// ---- VISUs/GlobalTextList_1.TcGTLO
TEXTLIST GlobalTextList_1
  2681 = '     '
  119 = '%' | German: '%' | France: '%' | English: '%'
  1446 = '%0.01f' | German: '%0.01f' | France: '%0.01f' | English: '%0.01f'
  4503 = '%0.02f' | German: '%0.02f' | France: '%0.02f' | English: '%0.02f'
  2738 = '%0.1f' | German: '%0.1f' | France: '%0.1f' | English: '%0.1f'
  537 = '%d' | German: '%d' | France: '%d' | English: '%d'
  890 = '%i' | German: '%i' | France: '%i' | English: '%i'
  1226 = '%i0.01f' | German: '%i0.01f' | France: '%i0.01f' | English: '%i0.01f'
  889 = '%s' | German: '%s' | France: '%s' | English: '%s'
  2909 = '(X100.00) STN 01 - 03 ULTRASONIC GENERATOR MCB - TRIP (-10F1)\n' | German: '(X100.00) WANNE 01 - WANNE 03 ULTRASCHALL GENERATOR SICHERUNG A AUSGELÖST (-10F1)' | France: '(X100.00) DEFAUT DISJONCTEUR GENE US POS 1 - POS 3 (-10F1)' | English: '(X100.00) STN 01 - 03 ULTRASONIC GENERATOR MCB - TRIP (-10F1)\n'
  3104 = '(X100.01) STN 01 ULTRASONIC GENERATOR (LEFT & RIGHT) - ALARM (-10U1)' | German: '(X100.01) WANNE 01 ULTRASCHALL GENERATOR (SEITE) SICHERUNG AUSGELÖST (-10U1)' | France: '(X100.01) CUVE 1 ALARME DU GENERATEUR ULTRASONS (COTE) (-10U1)' | English: '(X100.01) STN 01 ULTRASONIC GENERATOR (LEFT & RIGHT) - ALARM (-10U1)'
  9404 = '(X100.02) STN 01 ULTRASONIC GENERATOR (BOTTOM) - ALARM (-10U1)\n' | German: '(X100.02) WANNE 01 ULTRASCHALL GENERATOR (UNTEN) SICHERUNG AUSGELÖST (-10U1)' | France: '(X100.02) CUVE 2 ALARME DU GENERATEUR ULTRASONS (FOND) (-10U1)' | English: '(X100.02) STN 01 ULTRASONIC GENERATOR (BOTTOM) - ALARM (-10U1)\n'
  10481 = '(X100.03) STN 02 ULTRASONIC GENERATOR (LEFT & RIGHT) - ALARM (-10U1)\n' | German: '(X100.03) WANNE 02 ULTRASCHALL GENERATOR (SEITE) SICHERUNG AUSGELÖST (-10U1)' | France: '(X100.03) CUVE 2 ALARME DU GENERATEUR ULTRASONS (COTE) (-10U1)' | English: '(X100.03) STN 02 ULTRASONIC GENERATOR (LEFT & RIGHT) - ALARM (-10U1)\n'
  10488 = '(X100.04) STN 02 ULTRASONIC GENERATOR (BOTTOM) - ALARM (-10U1)\n' | German: '(X100.04) WANNE 02 ULTRASCHALL GENERATOR (UNTEN) SICHERUNG AUSGELÖST (-10U1)' | France: '(X100.04) CUVE 2 ALARME DU GENERATEUR ULTRASONS (FOND) (-10U1)' | English: '(X100.04) STN 02 ULTRASONIC GENERATOR (BOTTOM) - ALARM (-10U1)\n'
  5247 = '(X100.05) STN 03 ULTRASONIC GENERATOR (LEFT & RIGHT) - ALARM (-10U1)' | German: '(X100.05) WANNE 03 ULTRASCHALL GENERATOR (SEITE) SICHERUNG AUSGELÖST (-10U1)' | France: '(X100.05) CUVE 3 ALARME DU GENERATEUR ULTRASONS (COTE) (-10U1)' | English: '(X100.05) STN 03 ULTRASONIC GENERATOR (LEFT & RIGHT) - ALARM (-10U1)'
  11591 = '(X100.06) STN 03 ULTRASONIC GENERATOR (BOTTOM) - ALARM (-10U1)' | German: '(X100.06) WANNE 03 ULTRASCHALL GENERATOR (UNTEN) SICHERUNG AUSGELÖST (-10U1)' | France: '(X100.06) CUVE 3 ALARME DU GENERATEUR ULTRASONS (FOND) (-10U1)' | English: '(X100.06) STN 03 ULTRASONIC GENERATOR (BOTTOM) - ALARM (-10U1)'
  12139 = '(X100.07) STN 04 - 05 ULTRASONIC GENERATOR MCB - TRIP (-11F1)' | German: '(X100.07) WANNE 04 - WANNE 05 ULTRASCHALL GENERATOR SICHERUNG AUSGELÖST (-11F1)' | France: '(X100.07) DEFAUT DISJONCTEUR GENE US CUVE 4 - CUVE 5 (-11F1)' | English: '(X100.07) STN 04 - 05 ULTRASONIC GENERATOR MCB - TRIP (-11F1)'
  6933 = '(X100.08) STN 04 ULTRASONIC GENERATOR (LEFT & RIGHT) - ALARM (-11U1)' | German: '(X100.08) WANNE 04 ULTRASCHALL GENERATOR (SEITE) SICHERUNG AUSGELÖST (-11U1)' | France: '(X100.08) CUVE 4 ALARME DU GENERATEUR ULTRASONS (COTE) (-11U1)' | English: '(X100.08) STN 04 ULTRASONIC GENERATOR (LEFT & RIGHT) - ALARM (-11U1)'
  6619 = '(X100.09) STN 04 ULTRASONIC GENERATOR (BOTTOM) - ALARM (-11U1)' | German: '(X100.09) WANNE 04 ULTRASCHALL GENERATOR (UNTEN) SICHERUNG AUSGELÖST (-11U1)' | France: '(X100.09) CUVE 4 ALARME DU GENERATEUR ULTRASONS (FOND) (-11U1)' | English: '(X100.09) STN 04 ULTRASONIC GENERATOR (BOTTOM) - ALARM (-11U1)'
  4361 = '(X100.10) STN 05 ULTRASONIC GENERATOR (BOTTOM) - ALARM (-11U1)' | German: '(X100.10) WANNE 05 ULTRASCHALL GENERATOR (UNTEN) SICHERUNG AUSGELÖST (-11U1)' | France: '(X100.10) CUVE 5 ALARME DU GENERATEUR ULTRASONS (FOND) (-11U1)' | English: '(X100.10) STN 05 ULTRASONIC GENERATOR (BOTTOM) - ALARM (-11U1)'
  1199 = '(X100.11) GENERAL MAIN PANEL PB - E-STOP (-251S1)' | German: '(X100.11) HAUPTPANEL - NOT-AUS (-251S1)' | France: "(X100.11) ALARME ARRET D'URGENCE - BP PANEL (-251S1)" | English: '(X100.11) GENERAL MAIN PANEL PB - E-STOP (-251S1)'
  10185 = '(X100.12) OPERATOR PULL STRING - E-STOP (-251S2)' | German: '(X100.12) SICHERHEITSSEILZUG - NOT-AUS (-251S2)' | France: '(X100.12) DEFAUT BOUCLE ARRET URGENCE (-251S2)' | English: '(X100.12) OPERATOR PULL STRING - E-STOP (-251S2)'
  10087 = '(X100.13) MAINTENANCE PULL STRING - E-STOP  (-251S3)' | German: '(X100.13)WARTUNGSEILZUG NOT-AUS(-251S3)' | France: "(X100.13) CORDE D'ENTRETIEN - ARRÊT D'URGENCE (-251S3)" | English: '(X100.13) MAINTENANCE PULL STRING - E-STOP  (-251S3)'
  6489 = '(X100.14) GENERAL TOUCH MONITOR SOCKET ELCB - TRIP (-8Q1)' | German: '(X100.14) TOUCH SCREEN STECKDOSE SICHERUNG AUSGELÖST (-8Q1)' | France: '(X100.14) DEFAUT DISJONCTEUR PANEL OPERATEUR (-8Q1)' | English: '(X100.14) GENERAL TOUCH MONITOR SOCKET ELCB - TRIP (-8Q1)'
  7510 = '(X100.15) ARM 01 SERVO DRIVE MCB - TRIP (-40F1)' | German: '(X100.15) ARM 01 SERVO ANTRIEB MCB - AUSLÖSUNG (-40F1)' | France: '(X100.15) DEFAUT DISJONCTEUR SERVOMOTEUR ROBOT (-40F1)' | English: '(X100.15) ARM 01 SERVO DRIVE MCB - TRIP (-40F1)'
  11212 = '(X101.00) IPC DC ON SIGNAL (-410K1)' | German: '(X101.00) INDUSTRIE-PC GLEICHSTROM AUF SIGNAL (-410K1)' | France: '(X101.00)PC INDUSTRIEL COURANT CONTINU SUR SIGNAL(-410K1)' | English: '(X101.00) IPC DC ON SIGNAL (-410K1)'
  2968 = '(X101.01) PANEL VENTILATION FAN MCB - TRIP  (-6F1)\n' | German: '(X101.01) SCHALTSCHRANK VENTILATOR SICHERUNG AUSGELÖST  (-6F1)' | France: '(X101.01) DEFAUT DISJONCTEUR VENTILATEUR ARMOIRE ELECTRIQUE  (-6F1)' | English: '(X101.01) PANEL VENTILATION FAN MCB - TRIP  (-6F1)\n'
  9585 = '(X101.02) PANEL LIGHTING MCB - TRIP  (-5F1)' | German: '(X101.02) SCHALTSCHRANK BELEUCHTUNG SICHERUNG AUSGELÖST  (-5F1)' | France: '(X101.02) DEFAUT DISJONCTEUR ECLAIRAGE 1  (-5F1)' | English: '(X101.02) PANEL LIGHTING MCB - TRIP  (-5F1)'
  4159 = '(X101.03) MACHINE LIGHTING 01 MCB - TRIP (-5F2)' | German: '(X101.03) MASCHINENBELEUCHTUNG 01(-5F2)' | France: '(X101.03)ÉCLAIRAGE DE MACHINE 01(-5F2)' | English: '(X101.03) MACHINE LIGHTING 01 MCB - TRIP (-5F2)'
  7312 = '(X101.04) MACHINE LIGHTING 02 MCB - TRIP (-5F3)' | German: '(X101.04) MASCHINENBELEUCHTUNG 02(-5F3)' | France: '(X101.04)ÉCLAIRAGE DE MACHINE 02(-5F3)' | English: '(X101.04) MACHINE LIGHTING 02 MCB - TRIP (-5F3)'
  4346 = '(X101.05) GENERAL TOUCH MONITOR SOCKET MCB - TRIP (-8F1)' | German: '(X101.05) TOUCH SCREEN STECKDOSE SICHERUNG AUSGELÖST (-8F1)' | France: '(X101.05) DEFAUT DISJONCTEUR PANEL OPERATEUR (-8F1)' | English: '(X101.05) GENERAL TOUCH MONITOR SOCKET MCB - TRIP (-8F1)'
  8277 = '(X101.06) GENERAL PHASE SEQUENCE RELAY MCB - TRIP (-3F2)' | German: '(X101.06) DREHRICHTUNGSRELAIS SICHERUNG AUSGELÖST (-3F2)' | France: '(X101.06) DEFAUT DISJONCTEUR GENERAL (-3F2)' | English: '(X101.06) GENERAL PHASE SEQUENCE RELAY MCB - TRIP (-3F2)'
  9048 = '(X101.07) GENERAL PHASE SEQUENCE RELAY - TRIP (-3K1)' | German: '(X101.07) DREHRICHTUNGSRELAIS AUSGELÖST - ALARM (-3K1)' | France: '(X101.07) RELAIS ALARME  PHASE SEQUENCE (-3K1)' | English: '(X101.07) GENERAL PHASE SEQUENCE RELAY - TRIP (-3K1)'
  10253 = '(X101.08) STN 06 PROCESS TANK BLOWER MMS&TOR - TRIP (-100Q1)' | German: 'WANNE 06 PROZESS TANK GEBLÄSE MANUELLER MOTORSTARTER & THERMISCHE ÜBERLASTUNG AUSGELÖST' | France: 'CUVE 06 PROCESSUS RÉSERVOIR VENTILATEUR DÉMARRAGE MANUEL DU MOTEUR & SURCHARGE THERMIQUE DÉCLENCHÉE' | English: '(X101.08) STN 06 PROCESS TANK BLOWER MMS&TOR - TRIP (-100Q1)'
  5932 = '(X101.09) STN 01 - 06 EXHAUST BLOWER MMS&TOR - TRIP (-101Q1)' | German: 'WANNE 01 - 06 ABGASGEBLÄSE MANUELLER MOTORSTARTER & THERMISCHE ÜBERLASTUNG AUSGELÖST' | France: "CUVE 01 - 06 VENTILATEUR DE GAZ D'ÉCHAPPEMENT DÉMARRAGE MANUEL DU MOTEUR & SURCHARGE THERMIQUE DÉCLENCHÉE" | English: '(X101.09) STN 01 - 06 EXHAUST BLOWER MMS&TOR - TRIP (-101Q1)'
  6620 = '(X101.10) STN 01 - 05 AGITATION MOTOR MMS&TOR - TRIP (-160Q1)' | German: 'WANNE 01 - 05 MOTOR WARENBEWEGUNG MANUELLER MOTORSTARTER & THERMISCHE ÜBERLASTUNG AUSGELÖST' | France: 'CUVE 01 - 05 MOTEUR MOUVEMENT DU PRODUIT DÉMARREUR MANUEL DU MOTEUR & SURCHARGE THERMIQUE DÉCLENCHÉE' | English: '(X101.10) STN 01 - 05 AGITATION MOTOR MMS&TOR - TRIP (-160Q1)'
  5425 = '(X101.11) STN 01 DOSING PUMP MCB - TRIP (-70F1)' | German: '(X101.11) WANNE 01 DOSIERPUMPE SICHERUNG AUSGELÖST (-70F1)' | France: '(X101.11) CUVE 1 DEFAUT DISJONCTEUR POMPE DOSAGE (-70F1)' | English: '(X101.11) STN 01 DOSING PUMP MCB - TRIP (-70F1)'
  3137 = '(X101.12) STN 02 DOSING PUMP MCB - TRIP (-71F1)' | German: '(X101.12) WANNE 02 DOSIERPUMPE SICHERUNG AUSGELÖST (-71F1)' | France: '(X101.12) CUVE 2 DEFAUT DISJONCTEUR POMPE DOSAGE (-71F1)' | English: '(X101.12) STN 02 DOSING PUMP MCB - TRIP (-71F1)'
  3866 = '(X101.13) STN 03 DOSING PUMP MCB - TRIP (-72F1)' | German: '(X101.13) WANNE 03 DOSIERPUMPE SICHERUNG AUSGELÖST (-72F1)' | France: '(X101.13) CUVE 3 DEFAUT DISJONCTEUR POMPE DOSAGE (-72F1)' | English: '(X101.13) STN 03 DOSING PUMP MCB - TRIP (-72F1)'
  11364 = '(X101.14) STN 04 DOSING PUMP MCB - TRIP (-73F1)' | German: '(X101.14) WANNE 04 DOSIERPUMPE SICHERUNG AUSGELÖST (-73F1)' | France: '(X101.14) CUVE 4 DEFAUT DISJONCTEUR POMPE DOSAGE (-73F1)' | English: '(X101.14) STN 04 DOSING PUMP MCB - TRIP (-73F1)'
  8857 = '(X101.15) STN 01 DOSING CHEMICAL CONTAINER RELAY SIGNAL - FEEDBACK (-70K1)' | German: '(X101.15) WANNE 01 REINIGUNGSMITTELBEHÄLTER SENSOR 1 KONTAKTBLOCK - RÜCKMELDUNG (-70K1)' | France: '(X101.15) CUVE 1 DOSAGE RETOUR DU SIGNAL DU RELAIS DU CONTENEUR (-70K1)' | English: '(X101.15) STN 01 DOSING CHEMICAL CONTAINER RELAY SIGNAL - FEEDBACK (-70K1)'
  620 = '(X102.00) STN 01 PROCESS TANK PUMP MMS&TOR - TRIP (-74Q1)' | German: 'Wanne 01 Prozess Pumpe Tank Manueller Motorstarter & Thermische Überlastung Ausgelöst' | France: 'Cuve 01 Processus Pompe Réservoir Démarreur Manuel Du Moteur & Surcharge Thermique Déclenchée' | English: '(X102.00) STN 01 PROCESS TANK PUMP MMS&TOR - TRIP (-74Q1)'
  9751 = '(X102.01) STN 02 PROCESS TANK PUMP MMS&TOR - TRIP (-75Q1)' | German: 'Wanne 02 Prozess Pumpe Tank Manueller Motorstarter & Thermische Überlastung Ausgelöst' | France: 'Cuve 02 Processus Pompe Réservoir Démarreur Manuel Du Moteur & Surcharge Thermique Déclenchée' | English: '(X102.01) STN 02 PROCESS TANK PUMP MMS&TOR - TRIP (-75Q1)'
  11969 = '(X102.02) STN 03 PROCESS TANK PUMP MMS&TOR - TRIP (-76Q1)' | German: 'Wanne 03 Prozess Pumpe Tank Manueller Motorstarter & Thermische Überlastung Ausgelöst' | France: 'Cuve 03 Processus Pompe Réservoir Démarreur Manuel Du Moteur & Surcharge Thermique Déclenchée' | English: '(X102.02) STN 03 PROCESS TANK PUMP MMS&TOR - TRIP (-76Q1)'
  9673 = '(X102.03) STN 04 PROCESS TANK PUMP MMS&TOR - TRIP (-77Q1)' | German: 'Wanne 04 Prozess Pumpe Tank Manueller Motorstarter & Thermische Überlastung Ausgelöst' | France: 'Cuve 04 Processus Pompe Réservoir Démarreur Manuel Du Moteur & Surcharge Thermique Déclenchée' | English: '(X102.03) STN 04 PROCESS TANK PUMP MMS&TOR - TRIP (-77Q1)'
  4653 = '(X102.04) STN 05 PROCESS TANK PUMP MMS&TOR - TRIP (-78Q1)' | German: 'Wanne 05 Prozess Pumpe Tank Manueller Motorstarter & Thermische Überlastung Ausgelöst' | France: 'Cuve 05 Processus Pompe Réservoir Démarreur Manuel Du Moteur & Surcharge Thermique Déclenchée' | English: '(X102.04) STN 05 PROCESS TANK PUMP MMS&TOR - TRIP (-78Q1)'
  1689 = '(X102.05) STN 01 - 04 CHEMICAL RETURN TANK PUMP MMS&TOR - TRIP (-80Q1)' | German: 'Wanne 01 - 04 Pumpe Für Chemikalienrücklauftank Manueller Motoranlasser & Thermisches Überlastung Ausgelöst' | France: 'Cuve 01 - 04 Pompe Pour Réservoir De Retour De Produits Chimiques Démarreur Manuel Du Moteur & Relais Thermique De Surcharge Déclenché' | English: '(X102.05) STN 01 - 04 CHEMICAL RETURN TANK PUMP MMS&TOR - TRIP (-80Q1)'
  5529 = '(X102.06) STN 06 PROCESS TANK VACUUM PUMP MMS&TOR -TRIP (-79Q1)' | German: 'Wanne 06 Prozess Tank Vakuumpumpe Manueller Motorstarter & Thermische Überlastung Ausgelöst' | France: 'Cuve 06 Processus Réservoir Pompe À Vide Démarreur Manuel Du Moteur & Surcharge Thermique Déclenchée' | English: '(X102.06) STN 06 PROCESS TANK VACUUM PUMP MMS&TOR -TRIP (-79Q1)'
  315 = '(X102.07) STN 01 PROCESS TANK HEATER MCB - TRIP (-130F1)' | German: '(X102.07) WANNE 01 HEIZUNG SICHERUNG AUSGELÖST (-130F1)' | France: '(X102.07) CUVE 1 DEFAUT DISJONCTEUR CHAUFFAGE (-130F1)' | English: '(X102.07) STN 01 PROCESS TANK HEATER MCB - TRIP (-130F1)'
  910 = '(X102.08) STN 02 PROCESS TANK HEATER MCB - TRIP (-131F1)' | German: '(X102.08) WANNE 02 HEIZUNG SICHERUNG AUSGELÖST (-131F1)' | France: '(X102.08) CUVE 2 DEFAUT DISJONCTEUR CHAUFFAGE (-131F1)' | English: '(X102.08) STN 02 PROCESS TANK HEATER MCB - TRIP (-131F1)'
  6525 = '(X102.09) STN 03 PROCESS TANK HEATER MCB - TRIP (-132F1)' | German: '(X102.09) WANNE 03 HEIZUNG SICHERUNG AUSGELÖST (-132F1)' | France: '(X102.09) CUVE 3 DEFAUT DISJONCTEUR CHAUFFAGE (-132F1)' | English: '(X102.09) STN 03 PROCESS TANK HEATER MCB - TRIP (-132F1)'
  11585 = '(X102.10) STN 04 PROCESS TANK HEATER MCB - TRIP (-133F1)' | German: '(X102.10) WANNE 04 HEIZUNG SICHERUNG AUSGELÖST (-133F1)' | France: '(X102.10) CUVE 4 DEFAUT DISJONCTEUR CHAUFFAGE (-133F1)' | English: '(X102.10) STN 04 PROCESS TANK HEATER MCB - TRIP (-133F1)'
  3596 = '(X102.11) STN 06 PROCESS TANK HEATER MCB - TRIP (-134F1)' | German: '(X102.11) WANNE 06 HEIZUNG SICHERUNG AUSGELÖST (-134F1)' | France: '(X102.11) CUVE 6 DEFAUT DISJONCTEUR CHAUFFAGE (-134F1)' | English: '(X102.11) STN 06 PROCESS TANK HEATER MCB - TRIP (-134F1)'
  1057 = '(X102.12) LOADING CONVEYOR 1 MCB - TRIP (-170F1)' | German: '(X102.12) BELADEN FÖRDERBAND MOTOR 1 SICHERUNG AUSGELÖST (-170F1)' | France: '(X102.12) DISJONCTEUR CHARGEMENT MOTEUR CONV CHARG 1 (-170F1)' | English: '(X102.12) LOADING CONVEYOR 1 MCB - TRIP (-170F1)'
  11382 = '(X102.13) LOADING CONVEYOR 2 MCB - TRIP (-171F1)' | German: '(X102.13) BELADEN FÖRDERBAND MOTOR 2 SICHERUNG AUSGELÖST (-171F1)' | France: '(X102.13) DISJONCTEUR CHARGEMENT MOTEUR CONV CHARG 2 (-171F1)' | English: '(X102.13) LOADING CONVEYOR 2 MCB - TRIP (-171F1)'
  1453 = '(X102.14) LOADING CONVEYOR 3 MCB - TRIP (-172F1)' | German: '(X102.14) BELADEN FÖRDERBAND MOTOR 3 SICHERUNG AUSGELÖST (-172F1)' | France: '(X102.14) DISJONCTEUR CHARGEMENT MOTEUR CONV CHARG 3 (-172F1)' | English: '(X102.14) LOADING CONVEYOR 3 MCB - TRIP (-172F1)'
  1076 = '(X102.15) STN 02 DOSING CHEMICAL CONTAINER RELAY SIGNAL - FEEDBACK (-71K1)\n' | German: '(X102.15) WANNE 02 REINIGUNGSMITTELBEHÄLTER SENSOR 1 KONTAKTBLOCK - RÜCKMELDUNG (-71K1)' | France: '(X102.15) CUVE 2 DOSAGE RETOUR DU SIGNAL DU RELAIS DU CONTENEUR (-71K1)' | English: '(X102.15) STN 02 DOSING CHEMICAL CONTAINER RELAY SIGNAL - FEEDBACK (-71K1)\n'
  2864 = '(X103.00) MAIN SAFETY CONTACTOR 1 - FEEDBACK  (-250K1)' | German: '(X103.00) HAUPTSICHERHEITSSCHÜTZ 1 - RÜCKMELDUNG  (-250K1)' | France: '(X103.00) DEFAUT RETOUR CONTACTEUR GENERAL 1  (-250K1)' | English: '(X103.00) MAIN SAFETY CONTACTOR 1 - FEEDBACK  (-250K1)'
  3842 = '(X103.01) MAIN SAFETY CONTACTOR 2 - FEEDBACK  (-250K2)' | German: '(X103.01) HAUPTSICHERHEITSSCHÜTZ 2 - RÜCKMELDUNG  (-250K2)' | France: '(X103.01) DEFAUT RETOUR CONTACTEUR GENERAL 2  (-250K2)' | English: '(X103.01) MAIN SAFETY CONTACTOR 2 - FEEDBACK  (-250K2)'
  9985 = '(X103.02) DOOR SAFETY  CONTACTOR 1 - FEEDBACK  (-255K1)' | German: '(X103.02) TÜRSICHERHEITSSCHÜTZ 1 - RÜCKMELDUNG  (-255K1)' | France: '(X103.02) DEFAUT RETOUR CONTACTEUR SECURITE PORTE 1  (-255K1)' | English: '(X103.02) DOOR SAFETY  CONTACTOR 1 - FEEDBACK  (-255K1)'
  4912 = '(X103.03) DOOR SAFETY  CONTACTOR 2 - FEEDBACK  (-255K2)' | German: '(X103.03) TÜRSICHERHEITSSCHÜTZ 2 - RÜCKMELDUNG  (-255K2)' | France: '(X103.03) DEFAUT RETOUR CONTACTEUR SECURITE PORTE 2  (-255K2)' | English: '(X103.03) DOOR SAFETY  CONTACTOR 2 - FEEDBACK  (-255K2)'
  7342 = '(X103.04) MODULE 01 ADDITIONAL POWER SUPPLY INCOMING POWER MCB -TRIP (-4F3)\n' | German: '(X103.04)MODUL 01 ZUSÄTZLICHE STROMVERSORGUNG EINSPEISUNG SICHERUNG AUSGELÖST' | France: '(X103.04)MODUL 01 ZUSÄTZLICHE STROMVERSORGUNG EINSPEISUNG SICHERUNG AUSGELÖST' | English: '(X103.04) MODULE 01 ADDITIONAL POWER SUPPLY INCOMING POWER MCB -TRIP (-4F3)\n'
  8981 = '(X103.05) MODULE 01 ADDITIONAL POWER SUPPLY OUTGOING POWER MCB -TRIP (-4F4)' | German: '(X103.05)MODUL 01 ZUSÄTZLICHE STROMVERSORGUNG STROMAUSGANG SICHERUNG AUSGELÖST' | France: '(X103.05)MODULE 01 ALIMENTATION SUPPLÉMENTAIRE FUSIBLE DÉCLENCHÉE' | English: '(X103.05) MODULE 01 ADDITIONAL POWER SUPPLY OUTGOING POWER MCB -TRIP (-4F4)'
  2731 = '(X103.06) MODULE 02 ADDITIONAL POWER SUPPLY INCOMING POWER MCB -TRIP (-4F5)' | German: '(X103.06)MODUL 02 ZUSÄTZLICHE STROMVERSORGUNG EINSPEISUNG SICHERUNG AUSGELÖST' | France: '(X103.06)MODUL 02 ZUSÄTZLICHE STROMVERSORGUNG EINSPEISUNG SICHERUNG AUSGELÖST' | English: '(X103.06) MODULE 02 ADDITIONAL POWER SUPPLY INCOMING POWER MCB -TRIP (-4F5)'
  8822 = '(X103.07) MODULE 02 ADDITIONAL POWER SUPPLY OUTGOING POWER MCB -TRIP (-4F6)' | German: '(X103.07)MODUL 02 ZUSÄTZLICHE STROMVERSORGUNG STROMAUSGANG SICHERUNG AUSGELÖST' | France: '(X103.07)MODULE 02 ALIMENTATION SUPPLÉMENTAIRE FUSIBLE DÉCLENCHÉE' | English: '(X103.07) MODULE 02 ADDITIONAL POWER SUPPLY OUTGOING POWER MCB -TRIP (-4F6)'
  6849 = '(X103.08) MODULE 03 ADDITIONAL POWER SUPPLY INCOMING POWER MCB -TRIP (-4F7)' | German: '(X103.08)MODUL 03 ZUSÄTZLICHE STROMVERSORGUNG EINSPEISUNG SICHERUNG AUSGELÖST' | France: '(X103.08)MODUL 03 ZUSÄTZLICHE STROMVERSORGUNG EINSPEISUNG SICHERUNG AUSGELÖST' | English: '(X103.08) MODULE 03 ADDITIONAL POWER SUPPLY INCOMING POWER MCB -TRIP (-4F7)'
  3806 = '(X103.09) MODULE 03 ADDITIONAL POWER SUPPLY OUTGOING POWER MCB -TRIP (-4F8)' | German: '(X103.09)MODUL 03 ZUSÄTZLICHE STROMVERSORGUNG STROMAUSGANG SICHERUNG AUSGELÖST' | France: '(X103.09)MODULE 03 ALIMENTATION SUPPLÉMENTAIRE FUSIBLE DÉCLENCHÉE' | English: '(X103.09) MODULE 03 ADDITIONAL POWER SUPPLY OUTGOING POWER MCB -TRIP (-4F8)'
  2985 = '(X103.10) ARM 01 ADDITIONAL POWER SUPPLY INCOMING POWER MCB -TRIP (-4F9)' | German: '(X103.10)ROBOTER 01 ZUSÄTZLICHE STROMVERSORGUNG EINSPEISUNG SICHERUNG AUSGELÖST' | France: '(X103.10)ROBOT 01 ZUSÄTZLICHE STROMVERSORGUNG EINSPEISUNG SICHERUNG AUSGELÖST' | English: '(X103.10) ARM 01 ADDITIONAL POWER SUPPLY INCOMING POWER MCB -TRIP (-4F9)'
  4712 = '(X103.11) ARM 01 ADDITIONAL POWER SUPPLY OUTGOING POWER MCB -TRIP (-4F10)' | German: '(X103.11)ROBOTER 01 ZUSÄTZLICHE STROMVERSORGUNG STROMAUSGANG SICHERUNG AUSGELÖST' | France: '(X103.11)ROBOT 01 ALIMENTATION SUPPLÉMENTAIRE FUSIBLE DÉCLENCHÉE' | English: '(X103.11) ARM 01 ADDITIONAL POWER SUPPLY OUTGOING POWER MCB -TRIP (-4F10)'
  7888 = '(X103.12) STN 05 - 06 FFU UNIT MCB - TRIP (-163F1)' | German: '(X103.12)WANNE 05 - 06 VENTILATOR FILTER EINHEIT SICHERUNG AUSGELÖST' | France: '(X103.12)CUVE 05 - 06 UNITÉ VENTILATEUR FILTER FUSIBLE DÉCLENCHÉE' | English: '(X103.12) STN 05 - 06 FFU UNIT MCB - TRIP (-163F1)'
  12134 = '(X103.13) UNLOADING FFU UNIT MCB - TRIP (-164F1)' | German: '(X103.13)ENTLADEN FFU SICHERUNG AUSGELÖST' | France: '(X103.13)DECHARGEMET - UNITÉ VENTILATEUR FILTER FUSIBLE DÉCLENCHÉE' | English: '(X103.13) UNLOADING FFU UNIT MCB - TRIP (-164F1)'
  150 = '(X103.14) RESERVED' | German: '(X103.14)RESERVIERT' | France: '(X103.14)RESERVE' | English: '(X103.14) RESERVED'
  7835 = '(X103.15) RESERVED' | German: '(X103.15)RESERVIERT' | France: '(X103.15)RESERVE' | English: '(X103.15) RESERVED'
  4580 = '(X104.00) GENERAL ALARM PB - RESET (-304S1)' | German: '(X104.00) ALLGEMEINER ALARM PB - ZURÜCKSETZEN (-304S1)' | France: '(X104.00) RESET ALARM - BP RESET (-304S1)' | English: '(X104.00) GENERAL ALARM PB - RESET (-304S1)'
  12604 = '(X104.01) GENERAL BUZZER PB - RESET (-304S2)' | German: '(X104.01) ALLGEMEINER SUMMER PB - ZURÜCKSETZEN (-304S2)' | France: '(X104.01) RESET ALARM - BP ARRET BUZZER (-304S2)' | English: '(X104.01) GENERAL BUZZER PB - RESET (-304S2)'
  85 = '(X104.02) STN 01 PROCESS TANK SENSOR - MAX O/F (-304B1)' | German: 'WANNE 01 PROZESS TANK SENSOR - MAXIMALE ÜBERSCHREITUNG' | France: 'CUVE 01 CAPTEUR DE RÉSERVOIR DE TRAITEMENT - DÉBORDEMENT MAXIMAL' | English: '(X104.02) STN 01 PROCESS TANK SENSOR - MAX O/F (-304B1)'
  2048 = '(X104.03) STN 01 PROCESS TANK SENSOR - MIN O/F (-304B2)' | German: 'WANNE 01 PROZESS TANK SENSOR - MINIMALE ÜBERSCHREITUNG' | France: 'CUVE 01 CAPTEUR DE RÉSERVOIR DE TRAITEMENT - DÉBORDEMENT MINIMAL' | English: '(X104.03) STN 01 PROCESS TANK SENSOR - MIN O/F (-304B2)'
  9817 = '(X104.04) STN 01 PROCESS TANK SENSOR - MIN (-304B3)' | German: '(X104.04)  WANNE 01 NIVEAUSENSOR PROZESS - NIVEAU MINIMUM (-304B3)' | France: '(X104.04) CUVE 1 NIVEAU BAS (-304B3)' | English: '(X104.04) STN 01 PROCESS TANK SENSOR - MIN (-304B3)'
  527 = '(X104.05) STN 02 PROCESS TANK SENSOR - MAX O/F (-304B4)' | German: '(X104.05)WANNE 02 PROZESS TANK SENSOR - MAXIMALE ÜBERSCHREITUNG' | France: '(X104.05)CUVE 02 CAPTEUR DE RÉSERVOIR DE TRAITEMENT - DÉBORDEMENT MAXIMAL' | English: '(X104.05) STN 02 PROCESS TANK SENSOR - MAX O/F (-304B4)'
  4696 = '(X104.06) STN 02 PROCESS TANK SENSOR - MIN O/F (-304B5)' | German: '(X104.06) WANNE 02 PROZESS TANK SENSOR - MINIMALE ÜBERSCHREITUNG' | France: '(X104.06) CUVE 02 CAPTEUR DE RÉSERVOIR DE TRAITEMENT - DÉBORDEMENT MINIMAL' | English: '(X104.06) STN 02 PROCESS TANK SENSOR - MIN O/F (-304B5)'
  4065 = '(X104.07) STN 02 PROCESS TANK SENSOR - MIN (-304B6)' | German: '(X104.07)  WANNE 02 NIVEAUSENSOR PROZESS - NIVEAU MINIMUM (-304B6)' | France: '(X104.07) CUVE 2 NIVEAU BAS (-304B6)' | English: '(X104.07) STN 02 PROCESS TANK SENSOR - MIN (-304B6)'
  1186 = '(X104.08) STN 01 DOSING CHEMICAL CONTAINER SENSOR - WARNING LEVEL (-304S3)' | German: '(X104.08) WANNE 01 REINIGUNGSMITTELBEHÄLTER SENSOR 1 - NIVEAU WARNUNG (-304S3)' | France: '(X104.08) CUVE 1 AVERTISSEMENT DE NIVEAU MINI FUT LESSIVE DOSAGE (-304S3)' | English: '(X104.08) STN 01 DOSING CHEMICAL CONTAINER SENSOR - WARNING LEVEL (-304S3)'
  10163 = '(X104.09) STN 01 DOSING CHEMICAL CONTAINER SENSOR - MIN LEVEL (-304S3)' | German: '(X104.09) WANNE 01 REINIGUNGSMITTELBEHÄLTER SENSOR 1 - NIVEAU MINIMUM (-304S3)' | France: '(X104.09) CUVE 1 MINIMUM DE NIVEAU MINI FUT LESSIVE DOSAGE (-304S3)' | English: '(X104.09) STN 01 DOSING CHEMICAL CONTAINER SENSOR - MIN LEVEL (-304S3)'
  11193 = '(X104.10) STRUCTURE 01 DRIP PAN SENSOR - LEAK (-304B7)' | German: '(X104.10) STRUKTUR 1 LECKSENSOR - LECK (-304B7)' | France: '(X104.10) LA CARCASSE 1 FUITE LIQUIDE (-304B7)' | English: '(X104.10) STRUCTURE 01 DRIP PAN SENSOR - LEAK (-304B7)'
  12677 = '(X104.11) STN 02 DOSING CHEMICAL CONTAINER SENSOR - WARNING LEVEL (-304S4)' | German: '(X104.11) WANNE 02 REINIGUNGSMITTELBEHÄLTER SENSOR 1 - NIVEAU WARNUNG (-304S4)' | France: '(X104.11) CUVE 2 AVERTISSEMENT DE NIVEAU MINI FUT LESSIVE DOSAGE (-304S4)' | English: '(X104.11) STN 02 DOSING CHEMICAL CONTAINER SENSOR - WARNING LEVEL (-304S4)'
  10077 = '(X104.12) STN 02 DOSING CHEMICAL CONTAINER SENSOR - MIN LEVEL (-304S4)' | German: '(X104.12) WANNE 02 REINIGUNGSMITTELBEHÄLTER SENSOR 1 - NIVEAU MINIMUM (-304S4)' | France: '(X104.12) CUVE 2 MINIMUM DE NIVEAU MINI FUT LESSIVE DOSAGE (-304S4)' | English: '(X104.12) STN 02 DOSING CHEMICAL CONTAINER SENSOR - MIN LEVEL (-304S4)'
  4208 = '(X104.13) ARM 01 HORIZONTAL SENSOR - LOADING OT (-304B8)' | German: '(X104.13) ROBOTER 1 HORZ SENSOR - LADEN SEITE OT (-304B8)' | France: '(X104.13) SURCOURSE HORIZ RECUL  ROBOT1 (-304B8)' | English: '(X104.13) ARM 01 HORIZONTAL SENSOR - LOADING OT (-304B8)'
  2010 = '(X104.14) ARM 01 HORIZONTAL SENSOR - HOME (-304B9)' | German: '(X104.14) ROBOTER 1 HORZ SENSOR - LADEN SEITE HOME (-304B9)' | France: '(X104.14) DETECTEUR SYNCHRO ROBOT1 (-304B9)' | English: '(X104.14) ARM 01 HORIZONTAL SENSOR - HOME (-304B9)'
  6891 = '(X104.15) GENERAL SAFETY CURTAIN SENSOR - ALARM (-255K3)' | German: '(X104.15)ALLGEMEINER SICHERHEITSVORHANGSENSOR - ALARM' | France: '(X104.15)SÉCURITÉ GÉNÉRALE CAPTEUR DE RIDEAU - ALARME' | English: '(X104.15) GENERAL SAFETY CURTAIN SENSOR - ALARM (-255K3)'
  12989 = '(X110.00) ARM 01 VERTICAL SENSOR - TOP OT (-310B7)' | German: '(X110.00) ROBOTER 1 VERTIKAL SENSOR - OBEN TIMEOUT (-310B7)' | France: '(X110.00) DEFAUT FIN DE COURSE ROBOT 1 VERT (HAUT) (-310B7)' | English: '(X110.00) ARM 01 VERTICAL SENSOR - TOP OT (-310B7)'
  10651 = '(X110.01) ARM 01 VERTICAL SENSOR - HOME (-310B8)' | German: '(X110.01) ROBOTER 1 VERTIKAL SENSOR - OBEN NULLUNG (-310B8)' | France: '(X110.01) BRAS 1 ALARME DE MAISON VERTICALE COTE (-310B8)' | English: '(X110.01) ARM 01 VERTICAL SENSOR - HOME (-310B8)'
  7995 = '(X110.02) ARM 01 VERTICAL SENSOR - BTM OT (-310B9)' | German: '(X110.02) ROBOTER 1 VERTIKAL SENSOR - UNTEN TIMEOUT (-310B9)' | France: '(X110.02) DEFAUT VERT ROBOT 1 FIN DE COURSE (EN BAS) (-310B9)' | English: '(X110.02) ARM 01 VERTICAL SENSOR - BTM OT (-310B9)'
  9097 = '(X110.03) ARM 01 VERTICAL SENSOR - CRASH (-310B10)' | German: '(X110.03) ROBOTER 1 VERTIKAL SENSOR - AUFPRALL (-310B10)' | France: '(X110.03) DEFAUT SECURITE VERT ROBOT 1 (-310B10)' | English: '(X110.03) ARM 01 VERTICAL SENSOR - CRASH (-310B10)'
  4152 = '(X110.04) ARM 01 SENSOR A - MISSHOOK (-310B11)' | German: '(X110.04) ROBOTER 1 SENSOR A - FALSCHE BELEGUNG (-310B11)' | France: '(X110.04) DEFAUT ACCROCHAGE ROBOT 1 A (-310B11)' | English: '(X110.04) ARM 01 SENSOR A - MISSHOOK (-310B11)'
  5728 = '(X110.05) ARM 01 SENSOR B - MISSHOOK (-310B12)' | German: '(X110.05) ROBOTER 1 SENSOR B - FALSCHE BELEGUNG (-310B12)' | France: '(X110.05) DEFAUT ACCROCHAGE ROBOT 1 B (-310B12)' | English: '(X110.05) ARM 01 SENSOR B - MISSHOOK (-310B12)'
  10051 = '(X110.06) STN 03 PROCESS TANK SENSOR - MAX O/F (-310B1)' | German: '(X110.06)WANNE 03 PROZESS TANK SENSOR - MAXIMALE ÜBERSCHREITUNG' | France: '(X110.06)CUVE 03 CAPTEUR DE RÉSERVOIR DE TRAITEMENT - DÉBORDEMENT MAXIMAL' | English: '(X110.06) STN 03 PROCESS TANK SENSOR - MAX O/F (-310B1)'
  11634 = '(X110.07) STN 03 PROCESS TANK SENSOR - MIN O/F (-310B2)' | German: '(X110.07)WANNE 03 PROZESS TANK SENSOR - MINIMALE ÜBERSCHREITUNG' | France: '(X110.07)CUVE 03 CAPTEUR DE RÉSERVOIR DE TRAITEMENT - DÉBORDEMENT MINIMAL' | English: '(X110.07) STN 03 PROCESS TANK SENSOR - MIN O/F (-310B2)'
  362 = '(X110.08) STN 03 PROCESS TANK SENSOR - MIN (-310B3)' | German: '(X110.08)  WANNE 03 NIVEAUSENSOR PROZESS - NIVEAU MINIMUM (-310B3)' | France: '(X110.08) CUVE 3 DEFAUT NIVEAU BAS (-310B3)' | English: '(X110.08) STN 03 PROCESS TANK SENSOR - MIN (-310B3)'
  1438 = '(X110.09) STN 04 PROCESS TANK SENSOR - MAX O/F (-310B4)' | German: '(X110.09)WANNE 04 PROZESS TANK SENSOR - MAXIMALE ÜBERSCHREITUNG' | France: '(X110.09)CUVE 04 CAPTEUR DE RÉSERVOIR DE TRAITEMENT - DÉBORDEMENT MAXIMAL' | English: '(X110.09) STN 04 PROCESS TANK SENSOR - MAX O/F (-310B4)'
  11723 = '(X110.10) STN 04 PROCESS TANK SENSOR - MIN (-310B5)' | German: '(X110.10)  WANNE 04 NIVEAUSENSOR PROZESS - NIVEAU MINIMUM (-310B5)' | France: '(X110.10) CUVE 4 DEFAUT NIVEAU BAS (-310B5)' | English: '(X110.10) STN 04 PROCESS TANK SENSOR - MIN (-310B5)'
  10513 = '(X110.11) STRUCTURE 02 DRIP PAN SENSOR - LEAK (-310B6)' | German: '(X110.11) STRUKTUR 2 LECKSENSOR - LECK (-310B6)' | France: '(X110.11) LA CARCASSE 2 DEFAUT FUITE LIQUIDE (-310B6)' | English: '(X110.11) STRUCTURE 02 DRIP PAN SENSOR - LEAK (-310B6)'
  11762 = '(X110.12) STN 03 DOSING CHEMICAL CONTAINER SENSOR - WARNING LEVEL (-310S1)\n' | German: '(X110.12) WANNE 03 REINIGUNGSMITTELBEHÄLTER SENSOR 1 - NIVEAU WARNUNG (-310S1)' | France: '(X110.12) CUVE 3 AVERTISSEMENT DE NIVEAU MINI FUT LESSIVE DOSAGE (-310S1)' | English: '(X110.12) STN 03 DOSING CHEMICAL CONTAINER SENSOR - WARNING LEVEL (-310S1)\n'
  3924 = '(X110.13) STN 03 DOSING CHEMICAL CONTAINER SENSOR - MIN LEVEL (-310S1)' | German: '(X110.13) WANNE 03 REINIGUNGSMITTELBEHÄLTER SENSOR 1 - NIVEAU MINIMUM (-310S1)' | France: '(X110.13) CUVE 3 MINIMUM DE NIVEAU MINI FUT LESSIVE DOSAGE (-310S1)' | English: '(X110.13) STN 03 DOSING CHEMICAL CONTAINER SENSOR - MIN LEVEL (-310S1)'
  505 = '(X110.14) STN 04 DOSING CHEMICAL CONTAINER SENSOR - WARNING LEVEL (-310S2)' | German: '(X110.14) WANNE 04 REINIGUNGSMITTELBEHÄLTER SENSOR 1 - NIVEAU WARNUNG (-310S2)' | France: '(X110.14) CUVE 4 AVERTISSEMENT DE NIVEAU MINI FUT LESSIVE DOSAGE (-310S2)' | English: '(X110.14) STN 04 DOSING CHEMICAL CONTAINER SENSOR - WARNING LEVEL (-310S2)'
  11202 = '(X110.15) STN 04 DOSING CHEMICAL CONTAINER SENSOR - MIN LEVEL (-310S2)' | German: '(X110.15) WANNE 04 REINIGUNGSMITTELBEHÄLTER SENSOR 1 - NIVEAU MINIMUM (-310S2)' | France: '(X110.15) CUVE 4 MINIMUM DE NIVEAU MINI FUT LESSIVE DOSAGE (-310S2)' | English: '(X110.15) STN 04 DOSING CHEMICAL CONTAINER SENSOR - MIN LEVEL (-310S2)'
  1533 = '(X111.00) STN 03 DOSING CHEMICAL CONTAINER RELAY SIGNAL - FEEDBACK (-72K1)' | German: '(X111.00) WANNE 03 REINIGUNGSMITTELBEHÄLTER SENSOR 1 KONTAKTBLOCK - RÜCKMELDUNG (-72K1)' | France: '(X111.00) CUVE 3 DOSAGE RETOUR DU SIGNAL DU RELAIS DU CONTENEUR (-72K1)' | English: '(X111.00) STN 03 DOSING CHEMICAL CONTAINER RELAY SIGNAL - FEEDBACK (-72K1)'
  12520 = '(X111.01) STN 04 DOSING CHEMICAL CONTAINER RELAY SIGNAL - FEEDBACK (-73K1)' | German: '(X111.01) WANNE 04 REINIGUNGSMITTELBEHÄLTER SENSOR 1 KONTAKTBLOCK - RÜCKMELDUNG (-73K1)' | France: '(X111.01) CUVE 4 DOSAGE RETOUR DU SIGNAL DU RELAIS DU CONTENEUR (-73K1)' | English: '(X111.01) STN 04 DOSING CHEMICAL CONTAINER RELAY SIGNAL - FEEDBACK (-73K1)'
  4899 = '(X111.02) STN 04 PROCESS TANK SENSOR - MIN O/F (-311B1)' | German: '(X111.02)WANNE 04 PROZESS TANK SENSOR - MINIMALE ÜBERSCHREITUNG' | France: '(X111.02)CUVE 04 CAPTEUR DE RÉSERVOIR DE TRAITEMENT - DÉBORDEMENT MINIMAL' | English: '(X111.02) STN 04 PROCESS TANK SENSOR - MIN O/F (-311B1)'
  5642 = '(X111.03) RESERVED\n' | German: 'RESERVIERT' | France: 'RESERVE' | English: '(X111.03) RESERVED\n'
  3322 = '(X111.04) RESERVED' | German: 'RESERVIERT' | France: 'RESERVE' | English: '(X111.04) RESERVED'
  421 = '(X111.05) RESERVED' | German: 'RESERVIERT' | France: 'RESERVE' | English: '(X111.05) RESERVED'
  1655 = '(X111.06) RESERVED' | German: 'RESERVIERT' | France: 'RESERVE' | English: '(X111.06) RESERVED'
  9383 = '(X111.07) RESERVED' | German: 'RESERVIERT' | France: 'RESERVE' | English: '(X111.07) RESERVED'
  6156 = '(X111.08) RESERVED' | German: 'RESERVIERT' | France: 'RESERVE' | English: '(X111.08) RESERVED'
  9743 = '(X111.09) RESERVED\n' | German: 'RESERVIERT' | France: 'RESERVE' | English: '(X111.09) RESERVED\n'
  5314 = '(X111.10) RESERVED' | German: 'RESERVIERT' | France: 'RESERVE' | English: '(X111.10) RESERVED'
  3972 = '(X111.11) RESERVED\n' | German: 'RESERVIERT' | France: 'RESERVE' | English: '(X111.11) RESERVED\n'
  3844 = '(X111.12) RESERVED' | German: 'RESERVIERT' | France: 'RESERVE' | English: '(X111.12) RESERVED'
  636 = '(X111.13) RESERVED\n' | German: 'RESERVIERT' | France: 'RESERVE' | English: '(X111.13) RESERVED\n'
  2624 = '(X111.14) RESERVED\n' | German: 'RESERVIERT' | France: 'RESERVE' | English: '(X111.14) RESERVED\n'
  1246 = '(X111.15) RESERVED\n' | German: 'RESERVIERT' | France: 'RESERVE' | English: '(X111.15) RESERVED\n'
  4633 = '(X120.00) STN 05 PROCESS TANK SENSOR - MAX O/F (-320B1)' | German: '(X120.00)WANNE 05 PROZESS TANK SENSOR - MAXIMALE ÜBERSCHREITUNG' | France: '(X120.00)CUVE 05 CAPTEUR DE RÉSERVOIR DE TRAITEMENT - DÉBORDEMENT MAXIMAL' | English: '(X120.00) STN 05 PROCESS TANK SENSOR - MAX O/F (-320B1)'
  11874 = '(X120.01) STN 05 PROCESS TANK SENSOR - MIN (-320B2)' | German: '(X120.01)  WANNE 05 NIVEAUSENSOR PROZESS - NIVEAU MINIMUM (-320B2)' | France: '(X120.01) CUVE 5 DEFAUT NIVEAU BAS (-320B2)' | English: '(X120.01) STN 05 PROCESS TANK SENSOR - MIN (-320B2)'
  9495 = '(X120.02) STN 01 - 04 CHEMICAL RETURN TANK SENSOR - MAX (-320B3)' | German: '(X120.00)WANNE 01 - 04 SENSOR FÜR CHEMIKALIENRÜCKLAUFBEHÄLTER - MAXIMAL' | France: '(X120.00)CUVE 01 - 04 CAPTEUR DE RÉSERVOIR DE RETOUR DE PRODUITS CHIMIQUES - MAXIMUM' | English: '(X120.02) STN 01 - 04 CHEMICAL RETURN TANK SENSOR - MAX (-320B3)'
  9155 = '(X120.03) STN 01 - 04 CHEMICAL RETURN TANK SENSOR - REG (-320B4)' | German: '(X120.03)WANNE 01 - 04 SENSOR FÜR CHEMIKALIENRÜCKLAUFBEHÄLTER - SOLLWERT' | France: '(X120.03)CUVE 01 - 04 CAPTEUR DE RÉSERVOIR DE RETOUR DE PRODUITS CHIMIQUES - VALEUR DE CONSIGNE' | English: '(X120.03) STN 01 - 04 CHEMICAL RETURN TANK SENSOR - REG (-320B4)'
  10251 = '(X120.04) STN 01 - 04 CHEMICAL RETURN TANK SENSOR - MIN (-320B5)' | German: '(X120.04)WANNE 01 - 04 SENSOR FÜR CHEMIKALIENRÜCKLAUFBEHÄLTER - MINIMUM' | France: '(X120.04)CUVE 01 - 04 CAPTEUR DE RÉSERVOIR DE RETOUR DE PRODUITS CHIMIQUES - MINIMAL' | English: '(X120.04) STN 01 - 04 CHEMICAL RETURN TANK SENSOR - MIN (-320B5)'
  1697 = '(X120.05) STN 05 PROCESS TANK FLOW SENSOR - MIN FLOW (-320S1)' | German: '(X120.05)WANNE 05 PROZESS TANK DURCHFLUSSSENSOR - MINIMALDURCHFLUSS' | France: '(X120.05)CUVE 05 CAPTEUR DE DÉBIT DU RÉSERVOIR DE TRAITEMENT - DÉBIT MINIMUM' | English: '(X120.05) STN 05 PROCESS TANK FLOW SENSOR - MIN FLOW (-320S1)'
  3762 = '(X120.06) STN 06 PROCESS TANK HEATER THERMOSTAT - ALARM (-320S2)' | German: '(X120.06) WANNE 06 HEIZUNG THERMOSTAT - ALARM (-320S2)' | France: '(X120.06) DEFAUT CUVE 6 THERMOSTAT CHAUFFAGE (-120S3) (-320S2)' | English: '(X120.06) STN 06 PROCESS TANK HEATER THERMOSTAT - ALARM (-320S2)'
  10613 = '(X120.07) STN 06 SHUTTER DOOR RS - OPEN (-320S3)' | German: '(X120.07) WANNE 06 SCHIEBEDECKEL GEÖFFNET (-320S3)' | France: '(X120.07) COUVERCLE COULISSANT CUVE 6 OUV (-320S3)' | English: '(X120.07) STN 06 SHUTTER DOOR RS - OPEN (-320S3)'
  2184 = '(X120.08) STN 06 SHUTTER DOOR RS - CLOSE (-320S4)' | German: '(X120.08) WANNE 06 SCHIEBEDECKEL GESCHLOSSENE (-320S4)' | France: '(X120.08) COUVERCLE COULISSANT CUVE 6 FERM (-320S4)' | English: '(X120.08) STN 06 SHUTTER DOOR RS - CLOSE (-320S4)'
  7879 = '(X120.09) STRUCTURE 03 DRIP PAN SENSOR - LEAK (-320B6)' | German: '(X120.09) STRUKTUR 3 LECKSENSOR - LECK (-320B6)' | France: '(X120.09) LA CARCASSE 3 FUITE LIQUIDE (-320B6)' | English: '(X120.09) STRUCTURE 03 DRIP PAN SENSOR - LEAK (-320B6)'
  4230 = '(X120.10) GENERAL INCOMING CDA PRESSURE SWITCH - MIN PRESSURE (-320S5)' | German: '(X120.10) DRUCKLUFTSENSOR - DRUCK MINIMUM (-320S5)' | France: '(X120.10) ALIM AIR COMPRIME (-320S5)' | English: '(X120.10) GENERAL INCOMING CDA PRESSURE SWITCH - MIN PRESSURE (-320S5)'
  4949 = '(X120.11) UNLOADING SENSOR - BASKET DETECTION (-320B7)' | German: '(X120.11) ENTLADESENSOR - KORBERKENNUNG (-320B7)' | France: '(X120.11) CAPTEUR DE DÉCHARGEMENT - DÉTECTION DE PANIER (-320B7)' | English: '(X120.11) UNLOADING SENSOR - BASKET DETECTION (-320B7)'
  12570 = '(X120.12) ARM 01 HORIZONTAL SENSOR - UNLOADING OT (-320B8)' | German: '(X120.12) ROBOTER 1 HORZ SENSOR - SEITE TIMEOUT (-320B8)' | France: '(X120.12) SURCOURSE HORIZ AVANCE  ROBOT1 (-320B8)' | English: '(X120.12) ARM 01 HORIZONTAL SENSOR - UNLOADING OT (-320B8)'
  3635 = '(X120.13) RESERVED' | German: 'RESERVIERT' | France: 'RESERVE' | English: '(X120.13) RESERVED'
  2627 = '(X120.14) RESERVED' | German: 'RESERVIERT' | France: 'RESERVE' | English: '(X120.14) RESERVED'
  1145 = '(X120.15) RESERVED' | German: 'RESERVIERT' | France: 'RESERVE' | English: '(X120.15) RESERVED'
  7632 = '(X121.00) STN 06 SHUTTER DOOR RS 01 - CLAMP (-321S1)' | German: '(X121.00)WANNE 06 SCHIEBETÜR-REEDSCHALTER 01 - GESCHLOSSEN' | France: '(X121.00)CUVE 06 CAPTEUR PORTES COULISSANTES 01 - FERMÉ' | English: '(X121.00) STN 06 SHUTTER DOOR RS 01 - CLAMP (-321S1)'
  3825 = '(X121.01) STN 06 SHUTTER DOOR RS 01 - UNCLAMP (-321S2)' | German: '(X121.01)WANNE 06 SCHIEBETÜR-REEDSCHALTER 01 - GEÖFFNET' | France: '(X121.01)CUVE 06 CAPTEUR PORTES COULISSANTES 01 - OUVERT' | English: '(X121.01) STN 06 SHUTTER DOOR RS 01 - UNCLAMP (-321S2)'
  10015 = '(X121.02) STN 06 SHUTTER DOOR RS 02 - CLAMP (-321S3)' | German: '(X121.02)WANNE 06 SCHIEBETÜR-REEDSCHALTER 02 - GESCHLOSSEN' | France: '(X121.02)CUVE 06 CAPTEUR PORTES COULISSANTES 02 - FERMÉ' | English: '(X121.02) STN 06 SHUTTER DOOR RS 02 - CLAMP (-321S3)'
  615 = '(X121.03) STN 06 SHUTTER DOOR RS 02 - UNCLAMP (-321S4)\n' | German: '(X121.03) WANNE 06 SCHIEBETÜR-REEDSCHALTER 02 - GEÖFFNET' | France: '(X121.03) CUVE 06 CAPTEUR PORTES COULISSANTES 02 - OUVERT' | English: '(X121.03) STN 06 SHUTTER DOOR RS 02 - UNCLAMP (-321S4)\n'
  10327 = '(X121.04) RESERVED' | German: 'RESERVIERT' | France: 'RESERVE' | English: '(X121.04) RESERVED'
  2759 = '(X121.05) RESERVED' | German: 'RESERVIERT' | France: 'RESERVE' | English: '(X121.05) RESERVED'
  1035 = '(X121.07) RESERVED\n' | German: 'RESERVIERT' | France: 'RESERVE' | English: '(X121.07) RESERVED\n'
  12534 = '(X121.08) RESERVED\n' | German: 'RESERVIERT' | France: 'RESERVE' | English: '(X121.08) RESERVED\n'
  400 = '(X121.09) RESERVED' | German: 'RESERVIERT' | France: 'RESERVE' | English: '(X121.09) RESERVED'
  7041 = '(X121.10) RESERVED\n' | German: 'RESERVIERT' | France: 'RESERVE' | English: '(X121.10) RESERVED\n'
  13024 = '(X121.11) RESERVED' | German: 'RESERVIERT' | France: 'RESERVE' | English: '(X121.11) RESERVED'
  6920 = '(X121.12) RESERVED\n' | German: 'RESERVIERT' | France: 'RESERVE' | English: '(X121.12) RESERVED\n'
  2569 = '(X121.13) RESERVED\n' | German: 'RESERVIERT' | France: 'RESERVE' | English: '(X121.13) RESERVED\n'
  1238 = '(X121.14) RESERVED\n' | German: 'RESERVIERT' | France: 'RESERVE' | English: '(X121.14) RESERVED\n'
  4602 = '(X121.15) RESERVED\n' | German: 'RESERVIERT' | France: 'RESERVE' | English: '(X121.15) RESERVED\n'
  12780 = '(X12130.06) RESERVED' | German: 'RESERVIERT' | France: 'RESERVE' | English: '(X12130.06) RESERVED'
  6575 = '(X130.00) LOADING CONVEYOR SENSOR - FEED (-330B1)' | German: '(X130.00) BELADEN FÖRDERBAND SENSOR - LADEN (-330B1)' | France: '(X130.00) CHARGEMENT DEFAUT ALIM CAPTEUR CONV CHARG (-330B1)' | English: '(X130.00) LOADING CONVEYOR SENSOR - FEED (-330B1)'
  4551 = '(X130.01) LOADING CONVEYOR SENSOR - INDEX (-330B2)\n' | German: '(X130.01) BELADEN FÖRDERBAND SENSOR - INDEX (-330B2)' | France: '(X130.01) CHARGEMENT DEFAUT INDEX CAPTEUR CONV CHARG (-330B2)' | English: '(X130.01) LOADING CONVEYOR SENSOR - INDEX (-330B2)\n'
  12720 = '(X130.02) LOADING CONVEYOR SENSOR - PICK  (-330B3)' | German: '(X130.02) BELADEN FÖRDERBAND SENSOR - ENTLADEN  (-330B3)' | France: '(X130.02) CHARGEMENT DEFAUT CAPTEUR CONVOYEUR POSITION CHARG  (-330B3)' | English: '(X130.02) LOADING CONVEYOR SENSOR - PICK  (-330B3)'
  10446 = '(X130.03) GENERAL LOADING PB - E-STOP (-251S4)' | German: 'ALLGEMEINER LADEDRUCKKNOPF - NOT-AUS' | France: "BOUTON-POUSSOIR DE CHARGEMENT GÉNÉRAL - ARRÊT D'URGENCE" | English: '(X130.03) GENERAL LOADING PB - E-STOP (-251S4)'
  7225 = '(X130.04) RESERVED' | German: 'RESERVIERT' | France: 'RESERVE' | English: '(X130.04) RESERVED'
  2132 = '(X130.05) RESERVED\n' | German: 'RESERVIERT' | France: 'RESERVE' | English: '(X130.05) RESERVED\n'
  1761 = '(X130.06) RESERVED\n' | German: 'RESERVIERT' | France: 'RESERVE' | English: '(X130.06) RESERVED\n'
  4766 = '(X130.07) RESERVED' | German: 'RESERVIERT' | France: 'RESERVE' | English: '(X130.07) RESERVED'
  1698 = '(X130.08) RESERVED\n' | German: 'RESERVIERT' | France: 'RESERVE' | English: '(X130.08) RESERVED\n'
  3688 = '(X130.09) RESERVED\n' | German: 'RESERVIERT' | France: 'RESERVE' | English: '(X130.09) RESERVED\n'
  7104 = '(X130.10) RESERVED\n' | German: 'RESERVIERT' | France: 'RESERVE' | English: '(X130.10) RESERVED\n'
  1854 = '(X130.11) RESERVED\n' | German: 'RESERVIERT' | France: 'RESERVE' | English: '(X130.11) RESERVED\n'
  5960 = '(X130.12) RESERVED\n' | German: 'RESERVIERT' | France: 'RESERVE' | English: '(X130.12) RESERVED\n'
  4771 = '(X130.13) RESERVED\n' | German: 'RESERVIERT' | France: 'RESERVE' | English: '(X130.13) RESERVED\n'
  185 = '(X130.14) RESERVED\n' | German: 'RESERVIERT' | France: 'RESERVE' | English: '(X130.14) RESERVED\n'
  1144 = '(X130.15) RESERVED\n' | German: 'RESERVIERT' | France: 'RESERVE' | English: '(X130.15) RESERVED\n'
  9162 = '(Y100.00) EMERGENCY STOP SAFETY RELAY - RESET  (-250K3)\\' | France: '(Y100.00) REARMEMENT RELAIS DE SECURITE  (-250K3)' | English: '(Y100.00) EMERGENCY STOP SAFETY RELAY - RESET  (-250K3)\\'
  12386 = '(Y100.01) STN 01 - 03 ULTRASONIC GENERATOR FREQUENCY CHANGE BIT 1 (-10U1)' | German: 'WANNE 01 - 03 ULTRASCHALLGENERATOR FREQUENZÄNDERUNG BIT 1 (-10U1)' | France: "CUVE 01 - 03 CHANGEMENT DE FRÉQUENCE DU GÉNÉRATEUR D'ULTRASONS BIT 1" | English: '(Y100.01) STN 01 - 03 ULTRASONIC GENERATOR FREQUENCY CHANGE BIT 1 (-10U1)'
  9328 = '(Y100.02) STN 01 - 03 ULTRASONIC GENERATOR FREQUENCY CHANGE BIT 2 (-10U1)' | German: 'WANNE 01 - 03 ULTRASCHALLGENERATOR FREQUENZÄNDERUNG BIT 2 (-10U1)' | France: "CUVE 01 - 03 CHANGEMENT DE FRÉQUENCE DU GÉNÉRATEUR D'ULTRASONS BIT 2" | English: '(Y100.02) STN 01 - 03 ULTRASONIC GENERATOR FREQUENCY CHANGE BIT 2 (-10U1)'
  9208 = '(Y100.03) STN 04 - 05 ULTRASONIC GENERATOR FREQUENCY CHANGE BIT 1 (-11U1)' | German: 'WANNE 04 - 05 ULTRASCHALLGENERATOR FREQUENZÄNDERUNG BIT 1 (-10U1)' | France: "CUVE 04 - 05 CHANGEMENT DE FRÉQUENCE DU GÉNÉRATEUR D'ULTRASONS BIT 1" | English: '(Y100.03) STN 04 - 05 ULTRASONIC GENERATOR FREQUENCY CHANGE BIT 1 (-11U1)'
  3667 = '(Y100.04) STN 04 - 05 ULTRASONIC GENERATOR FREQUENCY CHANGE BIT 2 (-11U1)' | German: 'WANNE 04 - 05 ULTRASCHALLGENERATOR FREQUENZÄNDERUNG BIT 2 (-10U1)' | France: "CUVE 04 - 05 CHANGEMENT DE FRÉQUENCE DU GÉNÉRATEUR D'ULTRASONS BIT 2" | English: '(Y100.04) STN 04 - 05 ULTRASONIC GENERATOR FREQUENCY CHANGE BIT 2 (-11U1)'
  4791 = '(Y100.05) GENERAL ALARM RESET IND (-304S1)' | German: '(Y100.05) GENERELLER ANLAGENRESET (-304S1)' | France: '(Y100.05) RESET ALARME (-304S1)' | English: '(Y100.05) GENERAL ALARM RESET IND (-304S1)'
  6872 = '(Y100.06) GENERAL BUZZER  RESET IND (-304S2)' | German: '(Y100.06) ALLGEMEINER SUMMER ZURÜCKSETZEN (-304S2)' | France: '(Y100.06) RESET BUZZER (-304S2)' | English: '(Y100.06) GENERAL BUZZER  RESET IND (-304S2)'
  1691 = '(Y100.07) GENERAL BUZZER TONE 1 (-400H1)' | German: '(Y100.07) ALLGEMEINER SUMMERTON 1 (-400H1)' | France: '(Y100.07) BUZZER 1 (-400H1)' | English: '(Y100.07) GENERAL BUZZER TONE 1 (-400H1)'
  5301 = '(Y100.08) GENERAL BUZZER TONE 2 (-400H1)' | German: '(Y100.08) ALLGEMEINER SUMMERTON 2 (-400H1)' | France: '(Y100.08) BUZZER 2 (-400H1)' | English: '(Y100.08) GENERAL BUZZER TONE 2 (-400H1)'
  3358 = '(Y100.09) GENERAL TOWER LIGHT IND - RED (-400H2)' | German: '(Y100.09) AMPEL - ROT (-400H2)' | France: '(Y100.09) COLONNE LUMINEUSE ROUGE (-400H2)' | English: '(Y100.09) GENERAL TOWER LIGHT IND - RED (-400H2)'
  7213 = '(Y100.10) GENERAL TOWER LIGHT IND - YELLOW (-400H2)' | German: '(Y100.10) AMPEL - GELB (-400H2)' | France: '(Y100.10) COLONNE LUMINEUSE JAUNE (-400H2)' | English: '(Y100.10) GENERAL TOWER LIGHT IND - YELLOW (-400H2)'
  1059 = '(Y100.11) GENERAL TOWER LIGHT IND - GREEN (-400H2)' | German: '(Y100.11) AMPEL - GRÜN (-400H2)' | France: '(Y100.11) COLONNE LUMINEUSE VERT (-400H2)' | English: '(Y100.11) GENERAL TOWER LIGHT IND - GREEN (-400H2)'
  3384 = '(Y100.12) RESERVED(Y100.12) IPC DC ON HOLDING RELAY (-400K1)\n' | German: 'INDUSTRIE-PC GLEICHSTROM AUF HALTERELAIS ' | France: 'PC INDUSTRIEL COURANT CONTINU SUR RELAIS DE MAINTIEN ' | English: '(Y100.12) RESERVED(Y100.12) IPC DC ON HOLDING RELAY (-400K1)\n'
  1106 = '(Y100.13) STN 05 - 06 FFU UNIT ON/OFF ()' | German: 'WANNE 05 - 06 FILTER EINHEIT EIN/AUS' | France: 'CUVE 05 - 06 UNITÉ DE FILTRE ON/OFF' | English: '(Y100.13) STN 05 - 06 FFU UNIT ON/OFF ()'
  12934 = '(Y100.14) UNLOADING FFU UNIT ON/OFF ()' | German: 'ENTLADEN FILTER EINHEIT EIN/AUS' | France: 'DÉCHARGE UNITÉ DE FILTRE ON/OFF' | English: '(Y100.14) UNLOADING FFU UNIT ON/OFF ()'
  6399 = '(Y100.15) RESERVED\n' | German: 'RESERVIERT' | France: 'RESERVE' | English: '(Y100.15) RESERVED\n'
  10014 = '(Y101.00) STN 01 ULTRASONIC GENERATOR (LEFT &RIGHT) ON/OFF (-10U1)' | German: '(Y101.00) WANNE 01 ULTRASCHALLGENERATOREN (SEITE) EIN/AUS (-10U1)' | France: '(Y101.00) GENE US CUVE 1 (COTE) ON/OFF (-10U1)' | English: '(Y101.00) STN 01 ULTRASONIC GENERATOR (LEFT &RIGHT) ON/OFF (-10U1)'
  9375 = '(Y101.01) STN 01 ULTRASONIC GENERATOR (BOTTOM) ON/OFF (-10U1)' | German: '(Y101.01) WANNE 01 ULTRASCHALLGENERATOREN (UNTEN) EIN/AUS (-10U1)' | France: '(Y101.01) GENE US CUVE 1 (FOND) ON/OFF (-10U1)' | English: '(Y101.01) STN 01 ULTRASONIC GENERATOR (BOTTOM) ON/OFF (-10U1)'
  739 = '(Y101.02) STN 02 ULTRASONIC GENERATOR (LEFT &RIGHT) ON/OFF (-10U1)' | German: '(Y101.02) WANNE 02 ULTRASCHALLGENERATOREN (SEITE) EIN/AUS (-10U1)' | France: '(Y101.02) GENE US CUVE 2 (COTE) ON/OFF (-10U1)' | English: '(Y101.02) STN 02 ULTRASONIC GENERATOR (LEFT &RIGHT) ON/OFF (-10U1)'
  12798 = '(Y101.03) STN 02 ULTRASONIC GENERATOR (BOTTOM) ON/OFF (-10U1)' | German: '(Y101.03) WANNE 02 ULTRASCHALLGENERATOREN (UNTEN) EIN/AUS (-10U1)' | France: '(Y101.03) GENE US CUVE 2 (FOND) ON/OFF (-10U1)' | English: '(Y101.03) STN 02 ULTRASONIC GENERATOR (BOTTOM) ON/OFF (-10U1)'
  12492 = '(Y101.04) STN 03 ULTRASONIC GENERATOR (LEFT &RIGHT) ON/OFF (-10U1)' | German: '(Y101.04) WANNE 03 ULTRASCHALLGENERATOREN (SEITE) EIN/AUS (-10U1)' | France: '(Y101.04) GENE US CUVE 3 (COTE) ON/OFF (-10U1)' | English: '(Y101.04) STN 03 ULTRASONIC GENERATOR (LEFT &RIGHT) ON/OFF (-10U1)'
  9197 = '(Y101.05) STN 03 ULTRASONIC GENERATOR (BOTTOM) ON/OFF (-10U1)' | German: '(Y101.05) WANNE 03 ULTRASCHALLGENERATOREN (UNTEN) EIN/AUS (-10U1)' | France: '(Y101.05) GENE US CUVE 3 (FOND) ON/OFF (-10U1)' | English: '(Y101.05) STN 03 ULTRASONIC GENERATOR (BOTTOM) ON/OFF (-10U1)'
  12029 = '(Y101.06) STN 04 ULTRASONIC GENERATOR (LEFT &RIGHT) ON/OFF (-11U1)' | German: '(Y101.06) WANNE 04 ULTRASCHALLGENERATOREN (SEITE) EIN/AUS (-11U1)' | France: '(Y101.06) GENE US CUVE 4 (COTE) ON/OFF (-11U1)' | English: '(Y101.06) STN 04 ULTRASONIC GENERATOR (LEFT &RIGHT) ON/OFF (-11U1)'
  11238 = '(Y101.07) STN 04 ULTRASONIC GENERATOR (BOTTOM) ON/OFF (-11U1)' | German: '(Y101.07) WANNE 04 ULTRASCHALLGENERATOREN (UNTEN) EIN/AUS (-11U1)' | France: '(Y101.07) GENE US CUVE 4 (FOND) ON/OFF (-11U1)' | English: '(Y101.07) STN 04 ULTRASONIC GENERATOR (BOTTOM) ON/OFF (-11U1)'
  3974 = '(Y101.08) STN 05 ULTRASONIC GENERATOR (BOTTOM) ON/OFF (-11U1)' | German: '(Y101.08) WANNE 05 ULTRASCHALLGENERATOREN (UNTEN) EIN/AUS (-11U1)' | France: '(Y101.08) GENE US CUVE 5 (FOND) ON/OFF (-11U1)' | English: '(Y101.08) STN 05 ULTRASONIC GENERATOR (BOTTOM) ON/OFF (-11U1)'
  10864 = '(Y101.09) STN 01 DOSING PUMP ON/OFF (-70K1)' | German: '(Y101.09) WANNE 01 DOSIERPUMPE TANK EIN/AUS (-70K1)' | France: '(Y101.09) CUVE 1 POMPE DOSAGE ON/OFF (-70K1)' | English: '(Y101.09) STN 01 DOSING PUMP ON/OFF (-70K1)'
  2375 = '(Y101.10) STN 02 DOSING PUMP ON/OFF (-71K1)' | German: '(Y101.10) WANNE 02 DOSIERPUMPE TANK EIN/AUS (-71K1)' | France: '(Y101.10) CUVE 2 POMPE DOSAGE ON/OFF (-71K1)' | English: '(Y101.10) STN 02 DOSING PUMP ON/OFF (-71K1)'
  9806 = '(Y101.11) STN 01 PROCESS TANK PUMP ON/OFF (-74K1)' | German: '(Y101.11) WANNE 01 PROZESS TANK PUMPE EIN/AUS (-74K1)' | France: '(Y101.11) CUVE 1 POMPE ON/OFF (-74K1)' | English: '(Y101.11) STN 01 PROCESS TANK PUMP ON/OFF (-74K1)'
  11195 = '(Y101.12) STN 02 PROCESS TANK PUMP ON/OFF (-75K1)' | German: '(Y101.12) WANNE 02 PROZESS TANK PUMPE EIN/AUS (-75K1)' | France: '(Y101.12) CUVE 2 POMPE ON/OFF (-75K1)' | English: '(Y101.12) STN 02 PROCESS TANK PUMP ON/OFF (-75K1)'
  9429 = '(Y101.13) STN 03 PROCESS TANK PUMP ON/OFF (-76K1)' | German: '(Y101.13) WANNE 03 PROZESS TANK PUMPE EIN/AUS (-76K1)' | France: '(Y101.13) CUVE 3 POMPE ON/OFF (-76K1)' | English: '(Y101.13) STN 03 PROCESS TANK PUMP ON/OFF (-76K1)'
  12323 = '(Y101.14) STN 04 PROCESS TANK PUMP ON/OFF (-77K1)' | German: '(Y101.14) WANNE 04 PROZESS TANK PUMPE EIN/AUS (-77K1)' | France: '(Y101.14) CUVE 4 POMPE ON/OFF (-77K1)' | English: '(Y101.14) STN 04 PROCESS TANK PUMP ON/OFF (-77K1)'
  13519 = '(Y101.15) STN 05 PROCESS TANK PUMP ON/OFF (-78K1)' | German: '(Y101.15) WANNE 05 PROZESS TANK PUMPE EIN/AUS (-78K1)' | France: '(Y101.15) CUVE 5 POMPE ON/OFF (-78K1)' | English: '(Y101.15) STN 05 PROCESS TANK PUMP ON/OFF (-78K1)'
  2957 = '(Y102.00) STN 01 - 04 CHEMICAL RETURN TANK PUMP ON/OFF (-80K1)' | German: 'WANNE 01 - 04 PUMPE FÜR CHEMIKALIENRÜCKLAUFTANK EIN/AUS' | France: 'CUVE 01 - 04 POMPE DE RETOUR DE PRODUITS CHIMIQUES MARCHE/ARRÊT' | English: '(Y102.00) STN 01 - 04 CHEMICAL RETURN TANK PUMP ON/OFF (-80K1)'
  4102 = '(Y102.01) STN 06 PROCESS TANK VACUUM PUMP ON/OFF (-79K1)' | German: 'WANNE 06 PROZESSBEHÄLTER-VAKUUMPUMPE EIN/AUS' | France: 'CUVE 06 POMPE À VIDE MARCHE/ARRÊT' | English: '(Y102.01) STN 06 PROCESS TANK VACUUM PUMP ON/OFF (-79K1)'
  7047 = '(Y102.02) STN 01 PROCESS TANK HEATER ON/OFF (-130K1)' | German: '(Y102.02) WANNE 01 HEIZUNG TANK EIN/AUS (-130K1)' | France: '(Y102.02) CUVE 1 CHAUFFAGE ON/OFF (-130K1)' | English: '(Y102.02) STN 01 PROCESS TANK HEATER ON/OFF (-130K1)'
  11795 = '(Y102.03) STN 02 PROCESS TANK HEATER ON/OFF (-131K1)' | German: '(Y102.03) WANNE 02 HEIZUNG TANK EIN/AUS (-131K1)' | France: '(Y102.03) CUVE 2 CHAUFFAGE ON/OFF (-131K1)' | English: '(Y102.03) STN 02 PROCESS TANK HEATER ON/OFF (-131K1)'
  4147 = '(Y102.04) STN 03 PROCESS TANK HEATER ON/OFF (-132K1)' | German: '(Y102.04) WANNE 03 HEIZUNG TANK EIN/AUS (-132K1)' | France: '(Y102.04) CUVE 3 CHAUFFAGE ON/OFF (-132K1)' | English: '(Y102.04) STN 03 PROCESS TANK HEATER ON/OFF (-132K1)'
  1831 = '(Y102.05) STN 04 PROCESS TANK HEATER ON/OFF (-133K1)' | German: '(Y102.05) WANNE 04 HEIZUNG TANK EIN/AUS (-133K1)' | France: '(Y102.05) CUVE 4 CHAUFFAGE ON/OFF (-133K1)' | English: '(Y102.05) STN 04 PROCESS TANK HEATER ON/OFF (-133K1)'
  4645 = '(Y102.06) STN 06 PROCESS TANK HEATER ON/OFF (-134K1)' | German: '(Y102.06) WANNE 06 HEIZUNG TANK EIN/AUS (-134K1)' | France: '(Y102.06) CUVE 6 CHAUFFAGE ON/OFF (-134K1)' | English: '(Y102.06) STN 06 PROCESS TANK HEATER ON/OFF (-134K1)'
  1347 = '(Y102.07) STN 06 PROCESS TANK BLOWER ON/OFF (-100K1)' | German: '(Y102.07) WANNE 06 GEBLÄSE TROCKNER EIN/AUS (-100K1)' | France: '(Y102.07) CUVE 6 LE VENTILATEUR EST ON/OFF (-100K1)' | English: '(Y102.07) STN 06 PROCESS TANK BLOWER ON/OFF (-100K1)'
  8847 = '(Y102.08) STN 01 - 06 EXHAUST BLOWER ON/OFF (-101K1)' | German: 'WANNE 01 - 06 ABLUFTGEBLÄSE EIN/AUS' | France: "CUVE 01 - 06 VENTILATEUR D'EXTRACTION MARCHE/ARRÊT" | English: '(Y102.08) STN 01 - 06 EXHAUST BLOWER ON/OFF (-101K1)'
  11090 = '(Y102.09) RESERVED' | German: 'RESERVIERT' | France: 'RESERVE' | English: '(Y102.09) RESERVED'
  6826 = '(Y102.10) RESERVED\n' | German: 'RESERVIERT' | France: 'RESERVE' | English: '(Y102.10) RESERVED\n'
  9055 = '(Y102.11) RESERVED' | German: 'RESERVIERT' | France: 'RESERVE' | English: '(Y102.11) RESERVED'
  8987 = '(Y102.12) RESERVED' | German: 'RESERVIERT' | France: 'RESERVE' | English: '(Y102.12) RESERVED'
  1210 = '(Y102.13) RESERVED' | German: 'RESERVIERT' | France: 'RESERVE' | English: '(Y102.13) RESERVED'
  7178 = '(Y102.14) RESERVED\n' | German: 'RESERVIERT' | France: 'RESERVE' | English: '(Y102.14) RESERVED\n'
  3433 = '(Y102.15) RESERVED\n' | German: 'RESERVIERT' | France: 'RESERVE' | English: '(Y102.15) RESERVED\n'
  2494 = '(Y103.00) STN 01 - 05 AGITATION MOTOR ON/OFF (-160K1)' | German: '(Y103.00) WANNE 01-05 WARENBEWEGUNG MOTOR EIN/AUS (-160K1)' | France: '(Y103.00) CUVE 1-5 MOTEUR AGITATION ON/OFF (-160K1)' | English: '(Y103.00) STN 01 - 05 AGITATION MOTOR ON/OFF (-160K1)'
  7724 = '(Y103.01) LOADING CONVEYOR 01 ON/OFF (-170K1)' | German: '(Y103.01) BELADEN MOTOR FÖRDERBAND 1 EIN/AUS (-170K1)' | France: '(Y103.01) CHARGEMENT MOTEUR CONV CHARG 1 ON/OFF (-170K1)' | English: '(Y103.01) LOADING CONVEYOR 01 ON/OFF (-170K1)'
  12715 = '(Y103.02) LOADING CONVEYOR 02 ON/OFF (-171K1)' | German: '(Y103.02) BELADEN MOTOR FÖRDERBAND 2 EIN/AUS (-171K1)' | France: '(Y103.02) CHARGEMENT MOTEUR CONV CHARG 2 ON/OFF (-171K1)' | English: '(Y103.02) LOADING CONVEYOR 02 ON/OFF (-171K1)'
  500 = '(Y103.03) LOADING CONVEYOR 03 ON/OFF (-172K1)' | German: '(Y103.03) BELADEN MOTOR FÖRDERBAND 3 EIN/AUS (-172K1)' | France: '(Y103.03) CHARGEMENT MOTEUR CONV CHARG 3 ON/OFF (-172K1)' | English: '(Y103.03) LOADING CONVEYOR 03 ON/OFF (-172K1)'
  7713 = '(Y103.04) STATION ROTATION FOR ROTARY BARREL ON/OFF (-4K1 & 2)' | German: 'STATION DREHUNG FÜR DREHROHR EIN/AUS ' | France: "STATION DE ROTATION POUR L'ACTIVATION ET LA DÉSACTIVATION DU BARILLET ROTATIF " | English: '(Y103.04) STATION ROTATION FOR ROTARY BARREL ON/OFF (-4K1 & 2)'
  11682 = '(Y103.05) ROBOT ROTATION FOR ROTARY BARREL ON/OFF (-4K3)' | German: 'ROTATIONSROBOTER FÜR DAS EIN- UND AUSSCHALTEN DER TROMMEL' | France: "ROBOT DE ROTATION POUR L'ACTIVATION ET LA DÉSACTIVATION DU BARILLET ROTATIF" | English: '(Y103.05) ROBOT ROTATION FOR ROTARY BARREL ON/OFF (-4K3)'
  155 = '(Y103.06) RESERVED\n' | German: 'RESERVIERT' | France: 'RESERVE' | English: '(Y103.06) RESERVED\n'
  13498 = '(Y103.07) RESERVED\n' | German: 'RESERVIERT' | France: 'RESERVE' | English: '(Y103.07) RESERVED\n'
  12782 = '(Y103.08) RESERVED\n' | German: 'RESERVIERT' | France: 'RESERVE' | English: '(Y103.08) RESERVED\n'
  6048 = '(Y103.09) RESERVED\n' | German: 'RESERVIERT' | France: 'RESERVE' | English: '(Y103.09) RESERVED\n'
  1221 = '(Y103.10) RESERVED\n' | German: 'RESERVIERT' | France: 'RESERVE' | English: '(Y103.10) RESERVED\n'
  5649 = '(Y103.11) RESERVED\n' | German: 'RESERVIERT' | France: 'RESERVE' | English: '(Y103.11) RESERVED\n'
  8397 = '(Y103.12) RESERVED\n' | German: 'RESERVIERT' | France: 'RESERVE' | English: '(Y103.12) RESERVED\n'
  8137 = '(Y103.13) RESERVED\n' | German: 'RESERVIERT' | France: 'RESERVE' | English: '(Y103.13) RESERVED\n'
  5814 = '(Y103.14) RESERVED\n' | German: 'RESERVIERT' | France: 'RESERVE' | English: '(Y103.14) RESERVED\n'
  3911 = '(Y103.15) RESERVED\n' | German: 'RESERVIERT' | France: 'RESERVE' | English: '(Y103.15) RESERVED\n'
  6797 = '(Y110.00) STN 03 DOSING PUMP ON/OFF (-72K1)' | German: '(Y110.00) WANNE 03 DOSIERPUMPE TANK EIN/AUS (-72K1)' | France: '(Y110.00) CUVE 3 POMPE DOSAGE ON/OFF (-72K1)' | English: '(Y110.00) STN 03 DOSING PUMP ON/OFF (-72K1)'
  7268 = '(Y110.01) STN 04 DOSING PUMP ON/OFF (-73K1)' | German: '(Y110.01) WANNE 04 DOSIERPUMPE TANK EIN/AUS (-73K1)' | France: '(Y110.01) CUVE 4 POMPE DOSAGE ON/OFF (-73K1)' | English: '(Y110.01) STN 04 DOSING PUMP ON/OFF (-73K1)'
  8036 = '(Y110.02) RESERVED' | German: 'RESERVIERT' | France: 'RESERVE' | English: '(Y110.02) RESERVED'
  7206 = '(Y110.03) RESERVED' | German: 'RESERVIERT' | France: 'RESERVE' | English: '(Y110.03) RESERVED'
  10792 = '(Y110.04) RESERVED' | German: 'RESERVIERT' | France: 'RESERVE' | English: '(Y110.04) RESERVED'
  8398 = '(Y110.05) RESERVED' | German: 'RESERVIERT' | France: 'RESERVE' | English: '(Y110.05) RESERVED'
  1051 = '(Y110.06) RESERVED' | German: 'RESERVIERT' | France: 'RESERVE' | English: '(Y110.06) RESERVED'
  9996 = '(Y110.07) RESERVED' | German: 'RESERVIERT' | France: 'RESERVE' | English: '(Y110.07) RESERVED'
  6956 = '(Y110.08) RESERVED\n' | German: 'RESERVIERT' | France: 'RESERVE' | English: '(Y110.08) RESERVED\n'
  4075 = '(Y110.09) RESERVED\n' | German: 'RESERVIERT' | France: 'RESERVE' | English: '(Y110.09) RESERVED\n'
  2186 = '(Y110.10) RESERVED\n' | German: 'RESERVIERT' | France: 'RESERVE' | English: '(Y110.10) RESERVED\n'
  5827 = '(Y110.11) RESERVED\n' | German: 'RESERVIERT' | France: 'RESERVE' | English: '(Y110.11) RESERVED\n'
  271 = '(Y110.12) RESERVED\n' | German: 'RESERVIERT' | France: 'RESERVE' | English: '(Y110.12) RESERVED\n'
  3066 = '(Y110.13) RESERVED\n' | German: 'RESERVIERT' | France: 'RESERVE' | English: '(Y110.13) RESERVED\n'
  5337 = '(Y110.14) RESERVED\n' | German: 'RESERVIERT' | France: 'RESERVE' | English: '(Y110.14) RESERVED\n'
  5157 = '(Y110.15) RESERVED\n' | German: 'RESERVIERT' | France: 'RESERVE' | English: '(Y110.15) RESERVED\n'
  9394 = '(Y120.00) STN 01 INCOMING DIW SUPPLY AV1-1 (-420Y1)' | German: 'WANNE 01 EINGANG VERSORGUNG FÜR DEMINERALISIERTES WASSER LUFTVENTIL 1-1' | France: 'CUVE 01 ALIMENTATION EN EAU DÉMINÉRALISÉ' | English: '(Y120.00) STN 01 INCOMING DIW SUPPLY AV1-1 (-420Y1)'
  3345 = '(Y120.01) STN 01 OVERFLOW SUCTION AV1-2 (-420Y2)' | German: 'WANNE 01 ÜBERLAUF SAUGLUFTVENTIL 1-2' | France: "CUVE 01 SOUPAPE D'AIR D'ASPIRATION DE TROP-PLEIN 1-2" | English: '(Y120.01) STN 01 OVERFLOW SUCTION AV1-2 (-420Y2)'
  10197 = '(Y120.02) STN 01 BOTTOM SUCTION AV1-3 (-420Y3)' | German: 'WANNE 01 DRUCKTASTER SAUGLUFTVENTIL 1-3' | France: "CUVE 01 BOUTON-POUSSOIR SOUPAPE D'AIR D'ASPIRATION 1-3" | English: '(Y120.02) STN 01 BOTTOM SUCTION AV1-3 (-420Y3)'
  13660 = '(Y120.03) STN 01 DRAIN AV1-4 (-420Y4)' | German: 'WANNE 01 ENTLEERUNG SAUGLUFTVENTIL 1-4' | France: "CUVE 01 VIDANGE VANNE D'AIR D'ASPIRATION 1-4" | English: '(Y120.03) STN 01 DRAIN AV1-4 (-420Y4)'
  14091 = '(Y120.04) STN 02 INCOMING DIW SUPPLY AV2-1 (-420Y5)' | German: 'WANNE 02 EINGANG VERSORGUNG FÜR DEMINERALISIERTES WASSER LUFTVENTIL 2-1' | France: 'CUVE 02 ALIMENTATION EN EAU DÉMINÉRALISÉ' | English: '(Y120.04) STN 02 INCOMING DIW SUPPLY AV2-1 (-420Y5)'
  12279 = '(Y120.05) STN 02 OVERFLOW SUCTION AV2-2 (-420Y6)' | German: 'WANNE 02 ÜBERLAUF SAUGLUFTVENTIL 2-2' | France: "CUVE 02 SOUPAPE D'AIR D'ASPIRATION DE TROP-PLEIN 2-2" | English: '(Y120.05) STN 02 OVERFLOW SUCTION AV2-2 (-420Y6)'
  10215 = '(Y120.06) STN 02 BOTTOM SUCTION AV2-3 (-420Y7)' | German: 'WANNE 02 DRUCKTASTER SAUGLUFTVENTIL 2-3' | France: "CUVE 02 BOUTON-POUSSOIR SOUPAPE D'AIR D'ASPIRATION 2-3" | English: '(Y120.06) STN 02 BOTTOM SUCTION AV2-3 (-420Y7)'
  7352 = '(Y120.07) STN 02 DRAIN AV2-4 (-420Y8)' | German: 'WANNE 02 ENTLEERUNG SAUGLUFTVENTIL 2-4' | France: "CUVE 02 VIDANGE VANNE D'AIR D'ASPIRATION 2-4" | English: '(Y120.07) STN 02 DRAIN AV2-4 (-420Y8)'
  3939 = '(Y120.08) STN 03 INCOMING DIW SUPPLY AV3-1 (-420Y9)' | German: 'WANNE 03 EINGANG VERSORGUNG FÜR DEMINERALISIERTES WASSER LUFTVENTIL 3-1' | France: 'CUVE 03 ALIMENTATION EN EAU DÉMINÉRALISÉ' | English: '(Y120.08) STN 03 INCOMING DIW SUPPLY AV3-1 (-420Y9)'
  12053 = '(Y120.09) STN 03 OVERFLOW SUCTION AV3-2 (-420Y10)' | German: 'WANNE 03 ÜBERLAUF SAUGLUFTVENTIL 3-2' | France: "CUVE 03 SOUPAPE D'AIR D'ASPIRATION DE TROP-PLEIN 3-2" | English: '(Y120.09) STN 03 OVERFLOW SUCTION AV3-2 (-420Y10)'
  11532 = '(Y120.10) STN 03 BOTTOM SUCTION AV3-3 (-420Y11)' | German: 'WANNE 03 DRUCKTASTER SAUGLUFTVENTIL 3-3' | France: "CUVE 03 BOUTON-POUSSOIR SOUPAPE D'AIR D'ASPIRATION 3-3" | English: '(Y120.10) STN 03 BOTTOM SUCTION AV3-3 (-420Y11)'
  3310 = '(Y120.11) STN 03 DRAIN AV3-4 (-420Y12)' | German: 'WANNE 03 ENTLEERUNG SAUGLUFTVENTIL 3-4' | France: "CUVE 03 VIDANGE VANNE D'AIR D'ASPIRATION 3-4" | English: '(Y120.11) STN 03 DRAIN AV3-4 (-420Y12)'
  2986 = '(Y120.12) STN 04 INCOMING DIW SUPPLY AV4-1 (-420Y13)' | German: 'WANNE 04 EINGANG VERSORGUNG FÜR DEMINERALISIERTES WASSER LUFTVENTIL 4-1' | France: 'CUVE 04 ALIMENTATION EN EAU DÉMINÉRALISÉ' | English: '(Y120.12) STN 04 INCOMING DIW SUPPLY AV4-1 (-420Y13)'
  810 = '(Y120.13) STN 04 OVERFLOW SUCTION AV4-2 (-420Y14)' | German: 'WANNE 04 ÜBERLAUF SAUGLUFTVENTIL 4-2' | France: "CUVE 04 SOUPAPE D'AIR D'ASPIRATION DE TROP-PLEIN 4-2" | English: '(Y120.13) STN 04 OVERFLOW SUCTION AV4-2 (-420Y14)'
  2035 = '(Y120.14) STN 04 BOTTOM SUCTION AV4-3 (-420Y15)' | German: 'WANNE 04 DRUCKTASTER SAUGLUFTVENTIL 4-3' | France: "CUVE 04 BOUTON-POUSSOIR SOUPAPE D'AIR D'ASPIRATION 4-3" | English: '(Y120.14) STN 04 BOTTOM SUCTION AV4-3 (-420Y15)'
  6982 = '(Y120.15) STN 04 DRAIN AV4-4 (-420Y16)' | German: 'WANNE 04 ENTLEERUNG SAUGLUFTVENTIL 4-4' | France: "CUVE 04 VIDANGE VANNE D'AIR D'ASPIRATION 4-4" | English: '(Y120.15) STN 04 DRAIN AV4-4 (-420Y16)'
  13694 = '(Y121.00) STN 05 INCOMING DIW SUPPLY AV5-1 (-421Y1)' | German: 'WANNE 05 EINGANG VERSORGUNG FÜR DEMINERALISIERTES WASSER LUFTVENTIL 5-1' | France: 'CUVE 05 ALIMENTATION EN EAU DÉMINÉRALISÉ' | English: '(Y121.00) STN 05 INCOMING DIW SUPPLY AV5-1 (-421Y1)'
  5189 = '(Y121.01) STN 05 OVERFLOW SUCTION AV5-2 (-421Y2)' | German: 'WANNE 05 ÜBERLAUF SAUGLUFTVENTIL 5-2' | France: "CUVE 05 SOUPAPE D'AIR D'ASPIRATION DE TROP-PLEIN 5-2" | English: '(Y121.01) STN 05 OVERFLOW SUCTION AV5-2 (-421Y2)'
  5312 = '(Y121.02) STN 05 BOTTOM SUCTION AV5-3 (-421Y3)' | German: 'WANNE 05 DRUCKTASTER SAUGLUFTVENTIL 5-3' | France: "CUVE 05 BOUTON-POUSSOIR SOUPAPE D'AIR D'ASPIRATION 5-3" | English: '(Y121.02) STN 05 BOTTOM SUCTION AV5-3 (-421Y3)'
  7095 = '(Y121.03) STN 05 DRAIN AV5-4 (-421Y4)' | German: 'WANNE 05 ENTLEERUNG SAUGLUFTVENTIL 5-4' | France: "CUVE 05 VIDANGE VANNE D'AIR D'ASPIRATION 5-4" | English: '(Y121.03) STN 05 DRAIN AV5-4 (-421Y4)'
  13007 = '(Y121.04) STN 06 BLOWER PROTECTION AV6-1 (-421Y5)' | German: 'WANNE 06 GEBLÄSESCHUTZ SAUGLUFTVENTIL 6-1' | France: "CUVE 06 PROTECTION DU VENTILATEUR SOUPAPE D'AIR D'ASPIRATION 6-1" | English: '(Y121.04) STN 06 BLOWER PROTECTION AV6-1 (-421Y5)'
  3420 = '(Y121.05) STN 06 BLOWER PROTECTION AV6-2 (-421Y6)' | German: 'WANNE 06 GEBLÄSESCHUTZ SAUGLUFTVENTIL 6-2' | France: "CUVE 06 PROTECTION DU VENTILATEUR SOUPAPE D'AIR D'ASPIRATION 6-2" | English: '(Y121.05) STN 06 BLOWER PROTECTION AV6-2 (-421Y6)'
  1326 = '(Y121.06) STN 06 VACUUM SUCTION AV6-3 (-421Y7)' | German: 'WANNE 06 VAKUUMABSAUGUNG SAUGLUFTVENTIL 6-3' | France: "CUVE 06 ASPIRATION SOUS VIDE SOUPAPE D'AIR D'ASPIRATION 6-3" | English: '(Y121.06) STN 06 VACUUM SUCTION AV6-3 (-421Y7)'
  3917 = '(Y121.07) STN 06 VACUUM RELEASE AV6-4 (-421Y8)' | German: 'WANNE 06 VAKUUMENTLÜFTUNG SAUGLUFTVENTIL 6-4' | France: 'CUVE 06 VACUUM VENTILATION SUCTION AIR VALVE 6-4' | English: '(Y121.07) STN 06 VACUUM RELEASE AV6-4 (-421Y8)'
  9590 = '(Y121.08) GENERAL INCOMING DIW SUPPLY AVINC-1 (-421Y9)' | German: 'ALLGEMEINES EINSTRÖMENDES DIW-ZULUFTVENTIL INCOMING-1' | France: "VANNE D'ALIMENTATION EN AIR ENTRANT GÉNÉRAL DIW ENTRANT-1" | English: '(Y121.08) GENERAL INCOMING DIW SUPPLY AVINC-1 (-421Y9)'
  10324 = '(Y121.09) GENERAL INCOMING CW SUPPLY AVINC-2 (-421Y10)' | German: 'ALLGEMEINES EINSTRÖMENDES CW-ZULUFTVENTIL INCOMING-2' | France: "VANNE D'ALIMENTATION EN AIR ENTRANT GÉNÉRAL CW ENTRANT-2" | English: '(Y121.09) GENERAL INCOMING CW SUPPLY AVINC-2 (-421Y10)'
  525 = '(Y121.10) RESERVED\n' | German: 'RESERVIERT' | France: 'RESERVE' | English: '(Y121.10) RESERVED\n'
  6629 = '(Y121.11) RESERVED\n' | German: 'RESERVIERT' | France: 'RESERVE' | English: '(Y121.11) RESERVED\n'
  9736 = '(Y121.12) RESERVED\n' | German: 'RESERVIERT' | France: 'RESERVE' | English: '(Y121.12) RESERVED\n'
  5435 = '(Y121.13) RESERVED\n' | German: 'RESERVIERT' | France: 'RESERVE' | English: '(Y121.13) RESERVED\n'
  2693 = '(Y121.14) RESERVED\n' | German: 'RESERVIERT' | France: 'RESERVE' | English: '(Y121.14) RESERVED\n'
  8606 = '(Y121.15) RESERVED\n' | German: 'RESERVIERT' | France: 'RESERVE' | English: '(Y121.15) RESERVED\n'
  14346 = '(Y122.00) STN 06 SHUTTER DOOR - OPEN (-422Y1)' | German: '(Y122.00) WANNE 06 SCHIEBEDECKEL ÖFFNEN (-422Y1)' | France: '(Y122.00) COUVERCLE COULISSANT CUVE 6 OUV (-422Y1)' | English: '(Y122.00) STN 06 SHUTTER DOOR - OPEN (-422Y1)'
  10386 = '(Y122.01) STN 06 SHUTTER DOOR - CLOSE (-422Y2)\n' | German: '(Y122.01) WANNE 06 SCHIEBEDECKEL SCHLIESSEN (-422Y2)' | France: '(Y122.01) COUVERCLE COULISSANT CUVE 6 FERM (-422Y2)' | English: '(Y122.01) STN 06 SHUTTER DOOR - CLOSE (-422Y2)\n'
  7734 = '(Y122.02) STN 06 SHUTTER DOOR - CLAMP (-422Y3)\n' | German: 'WANNE 06 SCHIEBETÜRE GESCHLOSSEN' | France: 'CUVE 06 PORTE COULISSANTE FERMÉE' | English: '(Y122.02) STN 06 SHUTTER DOOR - CLAMP (-422Y3)\n'
  11353 = '(Y122.03) STN 06 SHUTTER DOOR - UNCLAMP (-422Y4)\n' | German: 'WANNE 06 SCHIEBETÜRE GEÖFFNET' | France: 'CUVE 06 PORTE COULISSANTE OUVERT' | English: '(Y122.03) STN 06 SHUTTER DOOR - UNCLAMP (-422Y4)\n'
  10729 = '(Y122.04) RESERVED\n' | German: 'RESERVIERT' | France: 'RESERVE' | English: '(Y122.04) RESERVED\n'
  13529 = '(Y122.05) RESERVED' | German: 'RESERVIERT' | France: 'RESERVE' | English: '(Y122.05) RESERVED'
  1773 = '(Y122.06) RESERVED' | German: 'RESERVIERT' | France: 'RESERVE' | English: '(Y122.06) RESERVED'
  5334 = '(Y122.07) RESERVED\n' | German: 'RESERVIERT' | France: 'RESERVE' | English: '(Y122.07) RESERVED\n'
  8088 = '(Y122.08) RESERVED\n' | German: 'RESERVIERT' | France: 'RESERVE' | English: '(Y122.08) RESERVED\n'
  5963 = '(Y122.09) RESERVED\n' | German: 'RESERVIERT' | France: 'RESERVE' | English: '(Y122.09) RESERVED\n'
  9740 = '(Y122.10) RESERVED\n' | German: 'RESERVIERT' | France: 'RESERVE' | English: '(Y122.10) RESERVED\n'
  1559 = '(Y122.11) RESERVED\n' | German: 'RESERVIERT' | France: 'RESERVE' | English: '(Y122.11) RESERVED\n'
  2852 = '(Y122.12) RESERVED\n' | German: 'RESERVIERT' | France: 'RESERVE' | English: '(Y122.12) RESERVED\n'
  3940 = '(Y122.13) RESERVED\n' | German: 'RESERVIERT' | France: 'RESERVE' | English: '(Y122.13) RESERVED\n'
  7536 = '(Y122.14) RESERVED\n' | German: 'RESERVIERT' | France: 'RESERVE' | English: '(Y122.14) RESERVED\n'
  4842 = '(Y122.15) RESERVED\n' | German: 'RESERVIERT' | France: 'RESERVE' | English: '(Y122.15) RESERVED\n'
  6003 = '1' | German: 'RESERVIERT' | France: 'RESERVE' | English: '1'
  3983 = '10' | German: '10' | France: '10' | English: '10'
  2050 = '11' | German: '11' | France: '11' | English: '11'
  3901 = '12' | German: '12' | France: '12' | English: '12'
  3843 = '13' | German: '13' | France: '13' | English: '13'
  909 = '14' | German: '14' | France: '14' | English: '14'
  1923 = '15' | German: '15' | France: '15' | English: '15'
  4708 = '16' | German: '16' | France: '16' | English: '16'
  2358 = '17' | German: '17' | France: '17' | English: '17'
  2692 = '18' | German: '18' | France: '18' | English: '18'
  2006 = '19' | German: '19' | France: '19' | English: '19'
  10521 = '1ST LIMIT ALARM (+/-)' | German: 'GRENZE 1 UBERSCHRITTEN AUSGELOST (+/-)' | France: '1ERE ALARME' | English: '1ST LIMIT ALARM (+/-)'
  1241 = '1st LIMIT TIMER' | German: '1. Grenzwerttimer' | France: '1. minuterie de limite' | English: '1st LIMIT TIMER'
  1993 = '1ST STAGE' | German: '1. STUFE' | France: '1POSITION' | English: '1ST STAGE'
  4717 = '1ST STAGE SPEED PROFILE' | German: '1. PHASE GESCHWINDIGKEITSPROFIL' | France: '1POSITION NIVEAU' | English: '1ST STAGE SPEED PROFILE'
  10596 = '1st VELO (mm/s)' | German: '1. GESCHIWINDIGKEIT (MM/S)' | France: '1POSITION VITESSE (mm/s)' | English: '1st VELO (mm/s)'
  5796 = '2' | German: '2' | France: '2' | English: '2'
  1058 = '20' | German: '20' | France: '20' | English: '20'
  112 = '21' | German: '21' | France: '21' | English: '21'
  7945 = '22' | German: '22' | France: '22' | English: '22'
  4534 = '23' | German: '23' | France: '23' | English: '23'
  3653 = '24' | German: '24' | France: '24' | English: '24'
  8275 = '25' | German: '25' | France: '25' | English: '25'
  410 = '26' | German: '26' | France: '26' | English: '26'
  9541 = '27' | German: '27' | France: '27' | English: '27'
  2771 = '28' | German: '28' | France: '28' | English: '28'
  4695 = '29' | German: '29' | France: '29' | English: '29'
  4466 = '2nd LIMIT TIMER' | German: '2. Grenzwerttimer' | France: '2. minuterie de limite' | English: '2nd LIMIT TIMER'
  5210 = '2ND STAGE' | German: '2. STUFE' | France: '2POSITION' | English: '2ND STAGE'
  5091 = '2ND STAGE SPEED PROFILE' | German: '2. PHASE GESCHWINDIGKEITSPROFIL' | France: '2POSITION NIVEAU' | English: '2ND STAGE SPEED PROFILE'
  3977 = '3' | German: '3' | France: '3' | English: '3'
  8083 = '30' | German: '30' | France: '30' | English: '30'
  7198 = '31' | German: '31' | France: '31' | English: '31'
  4660 = '32' | German: '32' | France: '32' | English: '32'
  6425 = '33' | German: '33' | France: '33' | English: '33'
  5399 = '34' | German: '34' | France: '34' | English: '34'
  5627 = '35' | German: '35' | France: '35' | English: '35'
  511 = '36' | German: '36' | France: '36' | English: '36'
  4805 = '37' | German: '37' | France: '37' | English: '37'
  2245 = '38' | German: '38' | France: '38' | English: '38'
  5102 = '39' | German: '39' | France: '39' | English: '39'
  2859 = '3RD STAGE' | German: '3. STUFE' | France: '3POSITION' | English: '3RD STAGE'
  2965 = '3RD STAGE SPEED PROFILE' | German: '3. PHASE GESCHWINDIGKEITSPROFIL' | France: '3POSITION NIVEAU' | English: '3RD STAGE SPEED PROFILE'
  5216 = '4' | German: '4' | France: '4' | English: '4'
  8783 = '40' | German: '40' | France: '40' | English: '40'
  2573 = '4TH STAGE' | German: '4. STUFE' | France: '4POSITION' | English: '4TH STAGE'
  1367 = '4TH STAGE SPEED PROFILE' | German: '4. PHASE GESCHWINDIGKEITSPROFIL' | France: '4POSITION NIVEAU' | English: '4TH STAGE SPEED PROFILE'
  6822 = '5' | German: '5' | France: '5' | English: '5'
  1400 = '6' | German: '6' | France: '6' | English: '6'
  6329 = '7' | German: '7' | France: '7' | English: '7'
  3152 = '7 DAYS PREPARATION' | German: '7D VORBEREITUNG' | France: '7D PREPARATION' | English: '7 DAYS PREPARATION'
  5104 = '8' | German: '8' | France: '8' | English: '8'
  7541 = '9' | German: '9' | France: '9' | English: '9'
  2450 = ':' | English: ':'
  591 = ': %0.01f' | German: ': %0.01f' | France: ': %0.01f' | English: ': %0.01f'
  1846 = 'ACC (mm/s2)' | German: 'ACC (mm/s2)' | France: 'ACC (mm/s2)' | English: 'ACC (mm/s2)'
  1228 = 'ACCESS LEVEL' | German: 'ZUGRIFFSEBENE' | France: "NIVEAU D'ACCÈS" | English: 'ACCESS LEVEL'
  2289 = 'ACTIVE ALARM' | German: 'AKTIV ALARM' | France: 'Alarme active' | English: 'ACTIVE ALARM'
  0 = 'ACTUAL VALUE' | German: 'TATSACHLICHER WERT' | France: 'TC REELLE' | English: 'ACTUAL VALUE'
  1966 = 'ADD USER' | German: 'BENUTZER\nHINZUFÜGEN' | France: 'AJOUTER UN\nUTILISATEUR' | English: 'ADD USER'
  58 = 'ALARM' | German: 'ALARM' | France: 'DEFAUT' | English: 'ALARM'
  2296 = 'ALARM HISTORY' | German: 'FEHLERHISTORIE' | France: "HISTORIQUE DE L'ALARME" | English: 'ALARM HISTORY'
  3527 = 'ALARM STATUS' | German: 'ALARM STATUS' | France: "ÉTAT DE L'ALARME" | English: 'ALARM STATUS'
  658 = 'ARM' | German: 'ROBOTER' | France: 'ROBOT' | English: 'ARM'
  1473 = 'Arm Busy' | German: 'ROBOTER BELEGT' | France: 'ROBOT OCCUPE' | English: 'Arm Busy'
  144 = 'ARM CONTROL' | German: 'ROBOTERKONTROLLE' | France: 'CONTRÔLE DES ROBOTS' | English: 'ARM CONTROL'
  502 = 'ARM HOMING :' | German: 'ROBOTER GRUNDSTELLUNG' | France: 'ROBOT POSITION DE BASE' | English: 'ARM HOMING :'
  2421 = 'ARM HORIZONTAL HOMING' | German: 'ROBOTER HORIZONTALE GRUNDSTELLUNG' | France: 'ROBOT POSITION DE BASE HORIZONTALE' | English: 'ARM HORIZONTAL HOMING'
  1701 = 'ARM HORIZONTAL POSITION (MM)' | German: 'ROBOTER HORIZONTALE POSITIONIERUNG' | France: 'ROBOT POSITIONNEMENT HORIZONTAL' | English: 'ARM HORIZONTAL POSITION (MM)'
  5912 = 'ARM HORIZONTAL SETTING' | German: 'HORIZONTALE EINSTELLUNG DES ARMS' | France: 'RÉGLAGE HORIZONTAL DU BRAS' | English: 'ARM HORIZONTAL SETTING'
  816 = 'ARM INFO' | German: 'ROBOTER DAS INFO' | France: 'ARM INFO' | English: 'ARM INFO'
  770 = 'ARM JOG VELO (mm/s)' | German: 'ROBOTER BEWEGUNG GESCHWINDIGKEIT (MM/S)' | France: 'ARM JOG VELO (mm/s)' | English: 'ARM JOG VELO (mm/s)'
  21 = 'ARM PATTERN' | German: 'ARM MUSTER' | France: 'MODÈLE DE BRAS' | English: 'ARM PATTERN'
  1169 = 'ARM POSITION' | German: 'ROBOTER POSITIONIERUNG' | France: 'POSITION DU BRAS' | English: 'ARM POSITION'
  5734 = 'ARM ROTATING ENABLE' | German: 'ROBOTER-DREHFREIGABE' | France: 'ACTIVATION DE LA ROTATION DU BRAS' | English: 'ARM ROTATING ENABLE'
  6770 = 'ARM ROTATION\nBASKET'
  6108 = 'ARM ROTATION BASKET'
  2637 = 'ARM SLOWPULL HOMING' | German: 'ROBOTER LIFT OUT GRUNDSTELLUNG' | English: 'ARM SLOWPULL HOMING'
  4587 = 'ARM SPEED PROFILE' | German: 'ROBOTER GESCHWINDIGKEIT PROFIL' | France: 'CONFIGURATION DES DIFFERENTES VITESSE DU ROBOT' | English: 'ARM SPEED PROFILE'
  670 = 'ARM STATUS' | German: 'ROBOTER STATUS' | France: 'ÉTAT DU BRAS' | English: 'ARM STATUS'
  2861 = 'ARM STN 1 UNHOOK' | German: 'ROBOTER WAHNE 1 AUSHANGEN' | France: 'ROBOT CUVE 1 DECROCHAGE' | English: 'ARM STN 1 UNHOOK'
  7281 = 'ARM UP' | German: 'ROBOTER ANFAHREN' | France: 'ROBOT HAUT' | English: 'ARM UP'
  2729 = 'ARM UP AND DOWN PATTERN' | German: 'ROBOTER OBEN UND UNTEN MUSTER' | France: 'CONFIGURATION DE LA VITESSE PAR POSITION' | English: 'ARM UP AND DOWN PATTERN'
  2463 = 'ARM VERTICAL HOMING' | German: 'ROBOTER VERTIKAL GRUNDSTELLUNG' | France: 'HOMING VERTICAL DU BRAS' | English: 'ARM VERTICAL HOMING'
  9150 = 'ARM VERTICAL POSITION (MM)' | German: 'ROBOTER VERTIKAL POSITION(mm)' | France: 'POSITION VERTICALE DU BRAS (MM)' | English: 'ARM VERTICAL POSITION (MM)'
  634 = 'ARM VERTICAL SETTING' | German: 'VERTICALE EINSTELLUNG DES ARMS' | France: 'RÉGLAGE VERTICAL DU BRAS' | English: 'ARM VERTICAL SETTING'
  3444 = 'ARM VERTICAL UP' | German: 'ROBOTER VERTIKAL ANFAHREN' | France: 'BRAS VERTICAL VERS LE HAUT' | English: 'ARM VERTICAL UP'
  365 = 'AUTO\nPREPARATION' | German: 'AUTO\nVORBEREITUNG' | France: 'PRÉPARATION\nAUTOMATIQUE' | English: 'AUTO\nPREPARATION'
  743 = 'AUTO MODE' | German: 'AUTO MODUS' | France: 'MODE AUTO' | English: 'AUTO MODE'
  722 = 'AUTO OPERATION SYSTEM CONTROL' | German: 'SYSTEMSTEUERUNG FÜR AUTOMATISCHEN BETRIEB' | France: 'CONTRÔLE DU SYSTÈME POUR UN FONCTIONNEMENT AUTOMATIQUE' | English: 'AUTO OPERATION SYSTEM CONTROL'
  911 = 'AUTO ORIGIN' | German: 'AUTO\nGRUNDSTELLUNG' | France: 'SYNCHRO ROBOT' | English: 'AUTO ORIGIN'
  1 = 'Auto Pre-Heat' | German: 'AUTO VORHEIZEN' | France: 'PRÉCHAUFFAGE AUTO' | English: 'Auto Pre-Heat'
  1117 = 'AUTO RUN' | German: 'AUTOMATIKBETRIEB' | France: 'MODE AUTOMATIQUE' | English: 'AUTO RUN'
  1837 = 'AUTO SHUTDOWN' | German: 'AUTOMATIKBETRIEB-AUSSCHALTEN' | France: 'DÉSACTIVATION DU MODE AUTOMATIQUE' | English: 'AUTO SHUTDOWN'
  369 = 'AUTO START' | German: 'AUTO START' | France: 'AUTO MODE' | English: 'AUTO START'
  5376 = 'BAD BASKET TOLERANCE TIME' | German: 'SCHLECHTE KORB TOLERANZZEIT' | France: 'MAUVAIS PANIER TEMPS DE TOLÉRANCE' | English: 'BAD BASKET TOLERANCE TIME'
  2857 = 'bar' | German: 'bar' | France: 'bar' | English: 'bar'
  3096 = 'Bar'
  310 = 'BARCODE' | German: 'BARCODE' | France: 'CODE À BARRE' | English: 'BARCODE'
  1080 = 'BARCODE\nENABLE' | German: 'BARCODE\nAKTIVIEREN' | France: 'CODE À BARRE\nACTIVER' | English: 'BARCODE\nENABLE'
  9047 = 'BARCODE\nPOPUP' | German: 'BARCODE\nPOPUP' | France: 'CODE À BARRE\nPOPUP' | English: 'BARCODE\nPOPUP'
  1558 = 'BARCODE / QR CODE' | German: 'BARCODE / QR CODE' | France: 'BARCODE / QR CODE' | English: 'BARCODE / QR CODE'
  5575 = 'BARCODE PAGE' | German: 'BARCODE-SEITE' | France: 'BARCODE CÔTÉ' | English: 'BARCODE PAGE'
  1313 = 'Barcode Received' | German: 'BARCODE SCAN' | France: 'LECTURE CODE BARRE' | English: 'Barcode Received'
  3624 = 'BARCODE REGISTER' | German: 'BARCODE-REGISTER' | France: 'BARCODE-REGISTER' | English: 'BARCODE REGISTER'
  344 = 'BARCODE REGISTRATION' | German: 'BARCODE-REGISTRIERUNG' | France: 'BARCODE ENREGISTREMENT' | English: 'BARCODE REGISTRATION'
  3053 = 'BARCODE STATUS' | German: 'BARCODE-STATUS' | France: 'BARCODE-STATUT' | English: 'BARCODE STATUS'
  2682 = 'BASIC' | German: 'GRUNDLEGENDE' | France: 'BASE' | English: 'BASIC'
  3887 = 'BASKET\nQUANTITY' | German: 'KORB MENGE' | France: 'NOMBRE DE PANIER' | English: 'BASKET\nQUANTITY'
  6885 = 'BASKET ID' | German: 'KORB-ID' | France: 'PANIER-ID' | English: 'BASKET ID'
  773 = 'BASKET QUANTITY' | German: 'KORB MENGE' | France: 'NOMBRE DE PANIER' | English: 'BASKET QUANTITY'
  3803 = 'BLOWER' | German: 'GEBLÄSE' | France: 'VENTILATEUR ' | English: 'BLOWER'
  3646 = 'BOTTOM POSITION' | German: 'POSITION UNTEN' | France: 'FOND DE CUVE' | English: 'BOTTOM POSITION'
  2931 = 'BUZZER\nRESET' | German: 'SUMMER\nZURUCKSETZEN' | France: 'RESET\nBUZZER' | English: 'BUZZER\nRESET'
  1856 = 'C' | German: 'C' | France: 'C' | English: 'C'
  1434 = 'CALIBRATE DONE' | German: 'KALIBRIEREN VOLLENDET' | France: 'CALIBRER' | English: 'CALIBRATE DONE'
  3324 = 'CALIBRATE FEED (pulse)' | German: 'BELADEN KALIBRIEREN' | France: 'CALIBRER ALIMENTATION' | English: 'CALIBRATE FEED (pulse)'
  285 = 'CALIBRATE IN PROGRESS' | German: 'KALIBRIERUNG LÄUFT' | France: 'ÉTALONNAGE EN COURS' | English: 'CALIBRATE IN PROGRESS'
  4915 = 'CALIBRATE RESULT (ml)' | German: 'KALIBRIERUNGSERGEBNIS (ml)' | France: 'RÉSULTAT DU CALIBRAGE (ml)' | English: 'CALIBRATE RESULT (ml)'
  4390 = 'CALIBRATE START' | German: 'KALIBRIEREN START' | France: 'CALIBRER DEMARRER' | English: 'CALIBRATE START'
  1774 = 'CALIBRATION' | German: 'KALIBRIEREN' | France: 'CALIBRER' | English: 'CALIBRATION'
  2503 = 'CANCEL' | German: 'ANNULIEREN' | France: 'ANNULER' | English: 'CANCEL'
  4131 = 'Cancel' | German: 'ANNULIEREN' | France: 'ANNULER' | English: 'Cancel'
  918 = 'CH' | German: 'CH' | France: 'CH' | English: 'CH'
  134 = 'CHANGE PASSWORD' | German: 'PASSWORD ANDERN' | France: 'CHANGER LE MOT DE PASSE' | English: 'CHANGE PASSWORD'
  2647 = 'CHANGE USER DETAILS AND INFORMATION' | German: 'BENUTZERDETAILS UND -INFORMATIONEN ÄNDERN' | France: "MODIFIER LES DÉTAILS ET LES INFORMATIONS DE L'UTILISATEUR" | English: 'CHANGE USER DETAILS AND INFORMATION'
  111 = 'CIRCULATION PUMP' | German: 'UMWALZPUMPE' | France: 'POMPE DE CIRCULATION' | English: 'CIRCULATION PUMP'
  1867 = 'CITY WATER SELECTION - AV 5-2' | German: 'UMWALZPUMPE' | France: 'POMPE DE CIRCULATION' | English: 'CITY WATER SELECTION - AV 5-2'
  6168 = 'CLAMP' | German: 'GESCHLOSSEN' | France: 'FERMÉ' | English: 'CLAMP'
  609 = 'CLEAR' | German: 'LÖSCHEN' | France: 'EFFACER' | English: 'CLEAR'
  6198 = 'CLOSE' | German: 'SCHLIESSEN' | France: 'FERME' | English: 'CLOSE'
  1340 = 'CONDUCTIVITY' | German: 'LEITFAHIGKET' | France: 'CONDUCTIVITE' | English: 'CONDUCTIVITY'
  943 = 'CONDUCTIVITY (μS)' | German: 'LEITFAHIGKET(μS)' | France: 'CONDUCTIVITE(μS)' | English: 'CONDUCTIVITY (μS)'
  4952 = 'CONFIG' | German: 'KONFIGURATION' | France: 'CONFIGURER' | English: 'CONFIG'
  1271 = 'CONFIRM' | German: 'BESTÄTIGEN' | France: 'CONFIRMER' | English: 'CONFIRM'
  791 = 'CONFIRM NEW PASSWORD' | German: 'NEUES PASSWORT BESTÄTIGEN' | France: 'CONFIRMER LE NOUVEAU MOT DE PASSE' | English: 'CONFIRM NEW PASSWORD'
  900 = 'COPY' | German: 'KOPIEREN' | France: 'COPIER' | English: 'COPY'
  2437 = 'COPY TO\nPROGRAM NO.' | German: 'IN PROGRAMM\nNR. KOPIEREN' | France: 'COPIER DANS LE\nPROGRAMME NO.' | English: 'COPY TO\nPROGRAM NO.'
  3155 = 'COPY TO PROGRAM NO.' | German: 'IN PROGRAMM NR. KOPIEREN' | France: 'COPIER DANS LE PROGRAMME NO.' | English: 'COPY TO PROGRAM NO.'
  2300 = 'CREATE\nUSER' | German: 'BENUTZER ERSTELLEN' | France: 'CRÉER UN UTILISATEUR' | English: 'CREATE\nUSER'
  102 = 'CREATE USER ACCOUNT TO GAIN CONTROL ACCESS' | German: 'BENUTZERKONTO ERSTELLEN\t UM KONTROLLZUGANG ZU ERHALTEN' | France: "CRÉER UN COMPTE D'UTILISATEUR POUR OBTENIR L'ACCÈS AU CONTRÔLE" | English: 'CREATE USER ACCOUNT TO GAIN CONTROL ACCESS'
  1958 = 'CURRENT PASSWORD' | German: 'AKTUELLES KENNWORT' | France: 'PENDANT  LE MOT DE PASSE' | English: 'CURRENT PASSWORD'
  4074 = 'CYCLE' | German: 'ZYKLUS' | France: 'CYCLE' | English: 'CYCLE'
  852 = 'DAILY' | German: 'TÄGLICH' | France: 'QUOTIDIENNEMENT' | English: 'DAILY'
  691 = 'DAY:HOUR:MIN:SEC' | German: 'TAG:STUNDE:MINUTE:SEKUNDE' | France: 'DATE : HEURE: MINUTE:' | English: 'DAY:HOUR:MIN:SEC'
  873 = 'DCC (mm/s2)' | German: 'abbremsen (mm/s2)' | France: 'DE’ACC (mm/s2)' | English: 'DCC (mm/s2)'
  493 = 'DEACTIVATED' | German: 'DEAKTIVIEREN' | France: 'DESACTIVER' | English: 'DEACTIVATED'
  2407 = 'DELAY TIME (s)' | German: 'VERZÖGERUNGSZEIT (s)' | France: "DÉLAI D'ATTENTE (sec.)" | English: 'DELAY TIME (s)'
  5460 = 'DELETE' | German: 'LÖSCHEN' | France: 'SUPPRIMER' | English: 'DELETE'
  1024 = 'DESCRIPTION' | German: 'BESCHREIBUNG' | France: 'DESCRIPTION' | English: 'DESCRIPTION'
  2820 = 'DI WATER SELECTION - AV 5-1' | English: 'DI WATER SELECTION - AV 5-1'
  3855 = 'DISABLE INSTRUMENT' | German: 'INSTRUMENT DEAKTIVIEREN' | France: 'INSTRUMENT DÉSACTIVER' | English: 'DISABLE INSTRUMENT'
  3225 = 'DISABLE INSTRUMENTS' | German: 'INSTRUMENT DEAKTIVIEREN' | France: 'INSTRUMENT DÉSACTIVER' | English: 'DISABLE INSTRUMENTS'
  2528 = 'DISABLE INSTRUMENTS AND ALARMS'
  346 = 'DIW MAIN INC AV-1' | German: 'DIONISATOR WASSER HAUPTZUFLUSS AV-1' | France: "VALVE D'AIR PRINCIPALE DE DIW INC-1" | English: 'DIW MAIN INC AV-1'
  610 = 'DO YOU WANT TO EXIT MANUAL MODE?' | German: 'SIND SIE SICHER\t DASS SIE DEN MANUELLEN MODUS VERLASSEN WOLLEN' | France: 'ETES VOUS SUR DE VOULOIR QUITTER LE MODE MANUEL' | English: 'DO YOU WANT TO EXIT MANUAL MODE?'
  4016 = 'DOOR' | German: 'SCHIEBTÜR' | France: 'PAR' | English: 'DOOR'
  6405 = 'DOOR CLAMP' | German: 'SCHIEBETÜRKLAMMER' | France: 'CLAMP DE PORTE' | English: 'DOOR CLAMP'
  4841 = 'DOOR CLOSE' | German: 'SCHIEBETÜR SCHLIESSEN' | France: 'PORTE FERMEE' | English: 'DOOR CLOSE'
  2846 = 'DOOR OPEN' | German: 'SCHIEBETÜR OFFEN' | France: 'PORTE OUVERTE' | English: 'DOOR OPEN'
  6495 = 'DOOR STN 6 CLAMP' | German: 'SCHIEBETÜR STN 6 KLAMMER' | France: 'À TRAVERS LE STN 6 CLAMP' | English: 'DOOR STN 6 CLAMP'
  3177 = 'DOOR STN 6 CLOSE' | German: 'SCHIEBETÜR STN 6 SCHLIESSEN' | France: 'À TRAVERS LE STN 6 FERMER' | English: 'DOOR STN 6 CLOSE'
  6487 = 'DOOR UNCLAMP' | German: 'SCHIEBETÜR ENTKLEMMEN' | France: 'PORTE DÉCROCHÉ' | English: 'DOOR UNCLAMP'
  8544 = 'DOSE PER PULSE (ml)' | German: 'DOSIERUNG PER PULSIEREN' | France: 'DOSAGE PAR PULSION' | English: 'DOSE PER PULSE (ml)'
  613 = 'DOSING' | German: 'DOSIERUNG' | France: 'DOSAGE' | English: 'DOSING'
  1538 = 'DOSING CALIBRATION' | German: 'DOSIERUNG KALIBRIEREN' | France: 'CALIBRATION DU DOSAGE' | English: 'DOSING CALIBRATION'
  1499 = 'DOWN' | German: 'EN BAS' | France: 'NACH UNTEN' | English: 'DOWN'
  2851 = 'DOWN TRANSFER' | German: 'NACH UNTEN TRANSFER' | France: 'CHOIX' | English: 'DOWN TRANSFER'
  5567 = 'DRIPPING TIME' | German: 'TROPEEN ZEIT' | France: 'TEMPS EGOUTTAGE' | English: 'DRIPPING TIME'
  3912 = 'EDIT' | German: 'BEARBEITEN' | France: 'EDIT' | English: 'EDIT'
  6373 = 'EDIT AND ADD USER'
  3660 = 'EDIT RECIPE' | German: 'REZEPT BEARBEITEN' | France: 'EDIT PROGRAMME' | English: 'EDIT RECIPE'
  4472 = 'ELAPSED TIME' | German: 'VERSTRICHENE ZEIT' | France: 'TEMPS ÉCOULÉ' | English: 'ELAPSED TIME'
  5466 = 'EN'
  7815 = 'ENABLE' | German: 'BEFAHIGEN' | France: 'ACTIVE' | English: 'ENABLE'
  357 = 'ENG' | German: 'ENG' | France: 'ENG' | English: 'ENG'
  355 = 'ENGINEER' | German: 'INGENIEUR' | France: 'INGENIEUR' | English: 'ENGINEER'
  838 = 'ERRORS AND WARNINGS' | German: 'FEHLER UND WARNUNGEN' | France: 'ERREURS ET AVERTISSEMENTS' | English: 'ERRORS AND WARNINGS'
  77 = 'EVENT\nRESET' | German: 'EREIGNIS\nZURÜCKSETZEN' | France: "RÉINITIALISATION\nDE L'ÉVÉNEMENT" | English: 'EVENT\nRESET'
  1859 = 'EVENT ID' | German: 'EREIGNIS ID' | France: 'ID ÉVÉNEMENT' | English: 'EVENT ID'
  3463 = 'FILTER' | German: 'FILTER' | France: 'FILTRE' | English: 'FILTER'
  4821 = 'FILTER PRESSURE (Bar)' | German: 'FILTERDRUCK(Bar)' | France: 'PRESSION DU FILTRE(Bar)' | English: 'FILTER PRESSURE (Bar)'
  767 = 'FILTER PRESSURE (bar)' | German: 'FILTERDRUCK(Bar)' | France: 'PRESSION DU FILTRE(Bar)' | English: 'FILTER PRESSURE (bar)'
  1253 = 'FIRST FILL (ml)' | German: 'ERSTE FULLEN' | France: 'PREMIER REMPLISSAGE' | English: 'FIRST FILL (ml)'
  1696 = 'FIRST NAME' | German: 'VORNAME' | France: 'PRÉNOM' | English: 'FIRST NAME'
  5450 = 'FR' | German: 'FR' | France: 'FR' | English: 'FR'
  6107 = 'FREQ' | German: 'FREQ' | France: 'FREQ' | English: 'FREQ'
  881 = 'FRI , 31MAR 2023 , 9:56:12 AM' | English: 'FRI , 31MAR 2023 , 9:56:12 AM'
  4621 = 'FRIDAY' | German: 'FREITAG' | France: 'VENDREDI' | English: 'FRIDAY'
  1542 = 'GENERAL INC CW AVINC-2' | German: 'ALLGEMEINES EINSTRÖMENDES CW-ZULUFTVENTIL INCOMING-2' | France: "VANNE D'ALIMENTATION EN AIR ENTRANT GÉNÉRAL CW ENTRANT-2" | English: 'GENERAL INC CW AVINC-2'
  4155 = 'GENERAL INC DIW AVINC-1' | German: 'ALLGEMEINES EINSTRÖMENDES DIW-ZULUFTVENTIL INCOMING-1' | France: "VANNE D'ALIMENTATION EN AIR ENTRANT GÉNÉRAL DIW ENTRANT-1" | English: 'GENERAL INC DIW AVINC-1'
  7132 = 'GENERAL INC DIW AVINC-2' | German: 'ALLGEMEINES EINSTRÖMENDES DIW-ZULUFTVENTIL INCOMING-2' | France: "VANNE D'ALIMENTATION EN AIR ENTRANT GÉNÉRAL DIW ENTRANT-2" | English: 'GENERAL INC DIW AVINC-2'
  1657 = 'GER' | German: 'DE' | France: 'DE' | English: 'GER'
  2876 = 'German' | German: 'Deutsch' | France: 'Deutsch' | English: 'German'
  3119 = 'HEATER' | German: 'HEIZUNG' | France: 'CHAUFFAGE' | English: 'HEATER'
  3092 = 'HIGH ALARM' | German: 'MAXIMALER ALARM' | France: 'ALARME MAXIMALE' | English: 'HIGH ALARM'
  203 = 'HIGH SAVE' | German: 'Hohen Wert speichern' | France: 'Enregistrer une valeur élevée' | English: 'HIGH SAVE'
  4356 = 'HIGH TEMP ALARM' | German: 'ALARM ÜBERTEMPERATUR' | France: 'ALARME DE TEMPÉRATURE ÉLEVÉE' | English: 'HIGH TEMP ALARM'
  8141 = 'High Vacuum Level' | German: 'HOHER VAKUUMGRAD' | France: 'HAUT NIVEAU DE SOUS-VIDE' | English: 'High Vacuum Level'
  6992 = 'HIGH VACUUM LEVEL' | German: 'HOHER VAKUUMGRAD' | France: 'HAUT NIVEAU DE SOUS-VIDE' | English: 'HIGH VACUUM LEVEL'
  2273 = 'HIGH VACUUM PRESSURE' | German: 'HOHER VAKUUMDRUCK ' | France: 'HAUTE PRESSION DU SOUS-VIDE' | English: 'HIGH VACUUM PRESSURE'
  2 = 'HOMING SECTION' | German: 'ROBOTER GRUNDSTELLUNG ABSCHNITT' | France: 'POINT SYNCHRO' | English: 'HOMING SECTION'
  2331 = 'HOOK' | German: 'HAKEN' | France: 'ACCROCHAGE' | English: 'HOOK'
  734 = 'HORIZONTAL' | German: 'HORIZONTALE' | France: 'HORIZONTALE' | English: 'HORIZONTAL'
  2378 = 'HOUR' | German: 'Stunde' | France: 'HEURE' | English: 'HOUR'
  3416 = 'HYSTERESIS' | German: 'HYSTERESIS' | France: 'HYSTERESIS' | English: 'HYSTERESIS'
  253 = 'I/O MONITORING' | German: 'IO UBERWACHUNG' | France: 'E/S VISUALISATION' | English: 'I/O MONITORING'
  703 = 'ID' | German: 'ID' | France: 'ID' | English: 'ID'
  3523 = 'INCOMING CITY WATER - AV 5-2'
  8167 = 'INCOMING DI WATER - AV 5-1'
  2254 = 'INCOMING VALVE DELAY OFF' | German: 'EINGANGSVENTILVERZÖGERUNG AUS' | France: "DÉLAI D'ARRÊT DE LA VANNE D'ENTRÉE" | English: 'INCOMING VALVE DELAY OFF'
  4371 = 'INPUT' | German: 'EINGABE' | France: 'ENTRÉE' | English: 'INPUT'
  3906 = 'IR HEATER TEMPERATURE (°C)' | German: 'IR-HEIZUNGSTEMPERATUR' | France: 'TEMPÉRATURE DU CHAUFFAGE IR' | English: 'IR HEATER TEMPERATURE (°C)'
  330 = 'JOG MODE' | German: 'JOG-BETRIEB' | France: 'TELECOMMANDE' | English: 'JOG MODE'
  600 = 'kHz' | German: 'kHz' | France: 'kHz' | English: 'kHz'
  316 = 'Kpa' | German: 'Kpa' | France: 'Kpa' | English: 'Kpa'
  4486 = 'kPa' | German: 'kPa' | France: 'kPa' | English: 'kPa'
  9520 = 'L' | German: 'L' | France: 'L' | English: 'L'
  830 = 'LANGUAGE :' | German: 'SPRACHE :' | France: 'LANGUE :' | English: 'LANGUAGE :'
  599 = 'LAST NAME' | German: 'NACHNAME' | France: 'NOM DE FAMILLE' | English: 'LAST NAME'
  2728 = 'LD\nDOWN' | German: 'LADE NACH\nUNTEN' | France: 'CHGT\nEN BAS' | English: 'LD\nDOWN'
  2158 = 'LD\nHOOK' | German: 'LADE NACH\nHAKEN' | France: 'CHGT\nACCROCHAGE' | English: 'LD\nHOOK'
  1638 = 'LD\nUNHOOK' | German: 'LADE NACH\nAUSHANGEN' | France: 'CHGT\nDECROCHAGE' | English: 'LD\nUNHOOK'
  1919 = 'LD CONVEYOR MOTOR 1' | German: 'BELADEN MOTOR\nFORDERBAND 01' | France: 'CHARGEMENT MOTEUR\nCONV CHARG 01' | English: 'LD CONVEYOR MOTOR 1'
  3077 = 'LD CONVEYOR MOTOR 2' | German: 'BELADEN MOTOR\nFORDERBAND 02' | France: 'CHARGEMENT MOTEUR\nCONV CHARG 02' | English: 'LD CONVEYOR MOTOR 2'
  3073 = 'LD CONVEYOR MOTOR 3' | German: 'BELADEN MOTOR\nFORDERBAND 03' | France: 'CHARGEMENT MOTEUR\nCONV CHARG 03' | English: 'LD CONVEYOR MOTOR 3'
  3022 = 'LD CONVEYOR MOTOR 4' | German: 'BELADEN MOTOR FORDERBAND 04' | France: 'CHARGEMENT MOTEUR CONV CHARG 04' | English: 'LD CONVEYOR MOTOR 4'
  4929 = 'LD CYCLINDER DOWN' | German: 'LADEZYLINDER UNTEN' | France: 'CYLINDRE DE CHARGEMENT EN BAS' | English: 'LD CYCLINDER DOWN'
  6576 = 'LD CYLINDER BACK' | German: 'LADEZYLINDER ZURÜCK' | France: 'CYLINDRE DE CHARGEMENT RETOUR' | English: 'LD CYLINDER BACK'
  2799 = 'LD CYLINDER BACK SESNOR' | German: 'LADEZYLINDER SENSOR ZURÜCK' | France: 'CYLINDRE DE CHARGEMENT CAPTEUR DE RETOUR' | English: 'LD CYLINDER BACK SESNOR'
  4138 = 'LD CYLINDER DOWN SENSOR' | German: 'LADEZYLINDER SENSOR UNTEN' | France: 'CYLINDRE DE CHARGEMENT CAPTEUR EN BAS' | English: 'LD CYLINDER DOWN SENSOR'
  3566 = 'LD CYLINDER FRONT' | German: 'LADEZYLINDER VORNE' | France: 'CYLINDRE DE CHARGEMENT AVANT' | English: 'LD CYLINDER FRONT'
  3593 = 'LD CYLINDER FRONT SENSOR' | German: 'LADEZYLINDER VORNE SENSOR' | France: 'CYLINDRE DE CHARGEMENT AVANT CAPTEUR' | English: 'LD CYLINDER FRONT SENSOR'
  4806 = 'LD CYLINDER UP' | German: 'LADEZYLINDER OBEN' | France: 'CYLINDRE DE CHARGEMENT EN HAUT' | English: 'LD CYLINDER UP'
  4463 = 'LD CYLINDER UP SESNOR' | German: 'LADEZYLINDER OBEN SENSOR' | France: 'CYLINDRE DE CHARGEMENT EN HAUT CAPTEUR' | English: 'LD CYLINDER UP SESNOR'
  2933 = 'LD MAX SENSOR' | German: 'LADEN MAXIMALER SENSOR' | France: 'CHARGEMENT CAPTEUR MAX' | English: 'LD MAX SENSOR'
  3711 = 'LD REG SENSOR' | German: 'LADEN DES REGULÄREN SENSORS' | France: 'CHARGEMENT CAPTEUR CONSIGNE' | English: 'LD REG SENSOR'
  1034 = 'LEFT\nBOTTOM' | German: 'LINKS UNTEN' | France: 'EN BAS À GAUCHE' | English: 'LEFT\nBOTTOM'
  1095 = 'LEFT\nTOP' | German: 'LINKS OBEN' | France: 'EN HAUT à GAUCHE' | English: 'LEFT\nTOP'
  2105 = 'LEFT BOTTOM TEMP (°C) ' | German: 'TEMPERATUR UNTEN LINKS' | France: 'TEMPÉRATURE EN BAS À GAUCHE' | English: 'LEFT BOTTOM TEMP (°C) '
  2616 = 'LEFT TOP TEMP (°C) ' | German: 'TEMPERATUR OBEN LINKS' | France: 'TEMPÉRATURE EN HAUT À GAUCHE' | English: 'LEFT TOP TEMP (°C) '
  916 = 'LEVEL' | German: 'STUFE' | France: 'NIVEAU' | English: 'LEVEL'
  1155 = 'LIST OF INPUTS AND OUTPUTS' | German: 'LISTE DER EIN- UND AUSGÄNGE' | France: 'LISTE DES ENTRÉES ET SORTIES' | English: 'LIST OF INPUTS AND OUTPUTS'
  3822 = 'Load basket'
  1138 = 'LOADING' | German: 'LADE' | France: 'CHARGEMENT' | English: 'LOADING'
  411 = 'LOG IN' | German: 'Anmeldung' | France: 'SE CONNECTER' | English: 'LOG IN'
  858 = 'LOG IN TO START OPERATE THE MACHINE' | German: 'ANMELDEN\t UM DIE MASCHINE ZU BETREIBEN' | France: 'SE CONNECTER POUR COMMENCER À UTILISER LA MACHINE' | English: 'LOG IN TO START OPERATE THE MACHINE'
  534 = 'LOG OUT' | German: 'AUSLOGGEN' | France: 'SE DECONNECTER' | English: 'LOG OUT'
  427 = 'LOG OUT OF SYSTEM' | German: 'AUS DEM SYSTEM AUSLOGGEN' | France: 'SE DÉCONNECTER DU SYSTÈME' | English: 'LOG OUT OF SYSTEM'
  7586 = 'Login Name' | German: 'ANMELDENAME' | France: 'NOM DE LOGIN' | English: 'Login Name'
  4330 = 'LOW ALARM' | German: 'NIEDRIGER ALARM' | France: 'BRAS BAS' | English: 'LOW ALARM'
  5373 = 'LOW SAVE' | German: 'Niedrigen Wert speichern' | France: 'Enregistrer une valeur basse' | English: 'LOW SAVE'
  1475 = 'Low Vacuum Level' | German: 'NIEDRIGES VAKUUM LEVEL' | France: 'BAS NIVEAU DE SOUS-VIDE' | English: 'Low Vacuum Level'
  1735 = 'LOW VACUUM LEVEL' | German: 'NIEDRIGES VAKUUM LEVEL' | France: 'BAS NIVEAU DE SOUS-VIDE' | English: 'LOW VACUUM LEVEL'
  7850 = 'LOW VACUUM PRESSURE' | German: 'NIEDERVAKUUMDRUCK' | France: 'BAS PRESSION DE SOUS-VIDE' | English: 'LOW VACUUM PRESSURE'
  1315 = 'MACHINE INFO' | German: 'MASCHINENINFORMATION' | France: 'INFORMATIONS SUR LA MACHINE' | English: 'MACHINE INFO'
  191 = 'MACHINE OPERATION HOUR          ' | German: 'MASCHINENBETRIEBSSTUNDE' | France: 'HEURE DE FONCTIONNEMENT\nDE LA MACHINE' | English: 'MACHINE OPERATION HOUR          '
  499 = 'MACHINE VIEW' | German: 'MASCHINENANSICHT' | France: 'VUE MACHINE' | English: 'MACHINE VIEW'
  242 = 'MAIN SYSTEM' | German: 'HAUPTSYSTEM' | France: 'MACHINE' | English: 'MAIN SYSTEM'
  762 = 'MAINTENANCE SYSTEM CONTROL' | German: 'STEUERUNG DES WARTUNGSSYSTEMS' | France: 'CONTRÔLE DU SYSTÈME DE MAINTENANCE' | English: 'MAINTENANCE SYSTEM CONTROL'
  3579 = 'MANUAL BASKET LOAD' | German: 'MANUELLE KORBBELADUNG' | France: 'CHARGEMENT MANUEL DU PANIER' | English: 'MANUAL BASKET LOAD'
  5048 = 'MANUAL DOSING' | German: 'MANUELL DOSIERUNG' | France: 'DOSAGE MANUEL' | English: 'MANUAL DOSING'
  1580 = 'MANUAL DOSING (ml)' | German: 'MANUELL DOSIERUNG (ml)' | France: 'DOSAGE MANUEL (ml)' | English: 'MANUAL DOSING (ml)'
  468 = 'MANUAL MODE' | German: 'HANDBUCH MODUS' | France: 'MODE MANUEL' | English: 'MANUAL MODE'
  1770 = 'MAXIMUM PROCESS TIME' | German: 'MAXIMALE PROZESSZEIT' | France: 'TEMPS MAXIMUM' | English: 'MAXIMUM PROCESS TIME'
  5270 = 'MID POSITION' | German: 'MITTLERE POSITION' | France: 'POSITION MÉDIANE' | English: 'MID POSITION'
  4416 = 'MINIMUM PROCESS TIME' | German: 'MINIMALE PROZESSKEIT' | France: 'TEMPS MINIMUM' | English: 'MINIMUM PROCESS TIME'
  460 = 'MINUTE' | German: 'Minute' | France: 'Minute' | English: 'MINUTE'
  1911 = 'ml' | German: 'ml' | France: 'ml' | English: 'ml'
  4815 = 'MONDAY' | German: 'Montag' | France: 'Lundi' | English: 'MONDAY'
  967 = 'N/A' | German: 'NICHT VERFÜGBAR' | France: 'NON DISPONIBLE' | English: 'N/A'
  2131 = 'N/A Load Time   :' | German: 'LADEZEIT NICHT VERFÜGBAR:' | France: 'NON DISPONIBLE TEMPS DE CHARGEMENT:' | English: 'N/A Load Time   :'
  241 = 'NEW PASSWORD' | German: 'NEUES KENNWORT' | France: 'NOUVEAU MOT DE PASSE' | English: 'NEW PASSWORD'
  1018 = 'NEW USER' | German: 'NEUER BENUTZER' | France: 'NOUVEL UTILISATEUR' | English: 'NEW USER'
  2698 = 'Next Load Time :' | German: 'Nächste Ladezeit :' | France: 'TEMPS DE CHARGEMENT SUIVANT' | English: 'Next Load Time :'
  5051 = 'NO' | German: 'Nummer' | France: 'Nombre' | English: 'NO'
  325 = 'NO.' | German: 'Nummer.' | France: 'Nombre.' | English: 'NO.'
  9420 = 'NOTICE !' | German: 'HINWEIS !' | France: 'REMARQUE' | English: 'NOTICE !'
  2535 = 'NUMBER OF BASKET\nBETWEEN DOSING' | German: 'ANZAHL DER KÖRBE ZWISCHEN DOSIERUNGEN' | France: 'NOMBRE DE PANIERS ENTRE LES DOSAGES' | English: 'NUMBER OF BASKET\nBETWEEN DOSING'
  1862 = 'OCCURRED' | German: 'EINGETRAGEN' | France: 'SURVENU' | English: 'OCCURRED'
  4569 = 'OFF' | German: 'ausschalten' | France: 'eteindre' | English: 'OFF'
  558 = 'OK' | German: 'OK' | France: 'OK' | English: 'OK'
  4314 = 'ON' | German: 'einschalten' | France: 'Allumer' | English: 'ON'
  313 = 'ORIGIN STATUS' | German: 'URSPRUNGSSTATUS' | France: "STATUT D'ORIGINE" | English: 'ORIGIN STATUS'
  1211 = 'OTHER INFO' | German: 'ANDERE INFORMATIONEN' | France: 'AUTRES INFORMATIONS' | English: 'OTHER INFO'
  7601 = 'OUTPUT' | German: 'AUSGANG' | France: 'SORTIE' | English: 'OUTPUT'
  1066 = 'OVERVIEW' | German: 'ÜBERSICHT' | France: 'APERÇU' | English: 'OVERVIEW'
  933 = 'PARAMETER' | German: 'PARAMETER' | France: 'PARAMÈTRE' | English: 'PARAMETER'
  1793 = 'PARAMETER\nOVERVIEW' | German: 'PARAMETERÜBERSICHT' | France: 'APERÇU DES PARAMÈTRES' | English: 'PARAMETER\nOVERVIEW'
  6578 = 'PARAMETER OVERVIEW' | German: 'PARAMETERÜBERSICHT' | France: 'APERÇU DES PARAMÈTRES' | English: 'PARAMETER OVERVIEW'
  840 = 'PASSWORD' | German: 'KENNWORT' | France: 'MODE POSSE' | English: 'PASSWORD'
  1633 = 'PICK & PLACE STATION ' | German: 'PICK & PLACE STATION ' | France: 'STATION PICK & PLACE ' | English: 'PICK & PLACE STATION '
  1474 = 'PICK UP' | German: 'ABHOLUNG' | France: 'PRENDRE' | English: 'PICK UP'
  2181 = 'Please key in recipe and press \nthe push button to load the basket' | German: 'Bitte geben Sie das Rezept ein und betätigen Sie die Drucktaste\t um den Korb zu laden.' | France: 'Veuillez saisir la recette et appuyer sur le bouton-poussoir pour charger le panier.' | English: 'Please key in recipe and press \nthe push button to load the basket'
  5474 = 'POSITION (mm)' | German: 'POSITION (mm)' | France: 'POSITION (MM)' | English: 'POSITION (mm)'
  2185 = 'POWER' | German: 'POWER' | France: 'POWER' | English: 'POWER'
  267 = 'POWER ON' | German: 'EINSCHALTEN' | France: 'MARCHE' | English: 'POWER ON'
  985 = 'PREPARATION STATUS' | German: 'VORBEREITUNGSSTAND' | France: 'ÉTAT DE PRÉPARATION' | English: 'PREPARATION STATUS'
  1556 = 'PRESSURE' | German: 'DRUCK' | France: 'PRESSION' | English: 'PRESSURE'
  1909 = 'PROCESS' | German: 'PROZESS' | France: 'PROCESSUS' | English: 'PROCESS'
  363 = 'PROCESS AND HANDLING PRESETS' | German: 'PROZESS- UND HANDHABUNGSVOREINSTELLUNGEN' | France: 'LES PRÉRÉGLAGES DE PROCESSUS ET DE TRAITEMENT' | English: 'PROCESS AND HANDLING PRESETS'
  48 = 'PROCESS MANAGEMENT' | German: 'PROZESSMANAGEMENT' | France: 'GESTION DES PROCESSUS' | English: 'PROCESS MANAGEMENT'
  314 = 'PROCESS STATUS' | German: 'PROZESSTATUS' | France: 'ETAT DU PROCESSUS' | English: 'PROCESS STATUS'
  3093 = 'PROCESS TANK' | German: 'PROZESS TANK' | France: 'CUVE DE TRAITEMENT' | English: 'PROCESS TANK'
  3650 = 'PROCESS TIME (s)' | German: 'PROZESS ZEIT (s)' | France: 'DUREE DU PROCESSUS (S)' | English: 'PROCESS TIME (s)'
  2438 = 'PROCESS TIME SV' | German: 'PROZESS ZEIT (SV)' | France: 'DUREE DU PROCESSUS (SV)' | English: 'PROCESS TIME SV'
  2980 = 'PRODUCT' | German: 'PRODUKT' | France: 'PRODUIT' | English: 'PRODUCT'
  478 = 'PRODUCT INFO' | German: 'PRODUKT-INFO' | France: 'INFORMATIONS SUR LE PRODUIT' | English: 'PRODUCT INFO'
  2493 = 'PRODUCT QUALITY' | German: 'PRODUKQUALITAT' | France: 'PRODUIT QUALITE' | English: 'PRODUCT QUALITY'
  2150 = 'PRODUCT RECIPE CONFIGURATION' | German: 'BESCHREIBUNG DES PRODUKTREZEPTS' | France: 'CONFIGURATION PROGRAMME PRODUIT' | English: 'PRODUCT RECIPE CONFIGURATION'
  539 = 'PRODUCT RECIPE DESCRIPTION' | German: 'REZEPTBESCHREIBUNG DES PRODUKTREZEPTS' | France: 'DESCRIPTION DE LA RECETTE DU PRODUIT' | English: 'PRODUCT RECIPE DESCRIPTION'
  4069 = 'PRODUCT RECIPE NO.' | German: 'PRODUKTREZEPTUR-NR.' | France: 'PROGRAMME PRODUIT NOMBRE' | English: 'PRODUCT RECIPE NO.'
  772 = 'PV' | German: 'AKTUELLER WERT' | France: 'ACTUEL' | English: 'PV'
  298 = 'QUALITY' | German: 'QUALITAT' | France: 'QUALITE' | English: 'QUALITY'
  10625 = 'READY (+/-)' | German: 'BEREIT(+/-)' | France: 'PRÊT(+/-)' | English: 'READY (+/-)'
  57 = 'RECIPE' | German: 'REZEPT' | France: 'PROGRAMME' | English: 'RECIPE'
  5669 = 'RECIPE DESCRIPTION' | German: 'REZEPTBESCHREIBUNG' | France: 'DESCRIPTION DE LA RECETTE' | English: 'RECIPE DESCRIPTION'
  283 = 'RECIPE NAME' | German: 'REZEPTNAME' | France: 'NOM DE LA RECETTE' | English: 'RECIPE NAME'
  941 = 'Recipe Name' | German: 'REZEPTNAME' | France: 'NOM DE LA RECETTE' | English: 'Recipe Name'
  2788 = 'RECIPE NO' | German: 'REZEPTNUMMER' | France: 'NUMERO DU PROGRAMME' | English: 'RECIPE NO'
  571 = 'RECIPE NO.' | German: 'REZEPTNUMMER' | France: 'NUMERO DU PROGRAMME' | English: 'RECIPE NO.'
  3419 = 'RECIPE OVERVIEW' | German: 'REZEPTÜBERSICHT' | France: 'APERÇU DES RECETTES' | English: 'RECIPE OVERVIEW'
  11375 = 'RECIPE PARAMETERS HAVE BEEN SAVED SUCCESSFULLY....' | German: 'DIE REZEPTPARAMETER WURDEN ERFOLGREICH GESPEICHERT....' | France: 'LES PARAMÈTRES DE LA RECETTE ONT ÉTÉ ENREGISTRÉS AVEC SUCCÈS....' | English: 'RECIPE PARAMETERS HAVE BEEN SAVED SUCCESSFULLY....'
  2776 = 'RECOVERED' | German: 'WIEDERHERGESTELLT' | France: 'RECOUVRÉ' | English: 'RECOVERED'
  7121 = 'REFERENCE MAXIMUM VACUUM READING' | German: 'MAXIMALER VAKUUMWERT - REFERENZ' | France: 'VALEUR MAXIMALE DU SOUS VIDE - RÉFÉRENCE' | English: 'REFERENCE MAXIMUM VACUUM READING'
  23 = 'REMAINING DOSING\nVOLUME (ml)' | German: 'Verbleibendes\nDosiervolumen (ml)' | France: 'DOSAGE\nNECESSAIRE (ML)' | English: 'REMAINING DOSING\nVOLUME (ml)'
  453 = 'REPEAT FROM\nSTEP NO.' | German: 'AB SCHRITT NR. WIEDERHOLEN.' | France: "RÉPÉTER À PARTIR DE L'ÉTAPE N°." | English: 'REPEAT FROM\nSTEP NO.'
  1893 = 'Reset' | German: 'ZURUCKSETZEN' | France: 'Remise a Zero' | English: 'Reset'
  1007 = 'RESET' | German: 'ZURUCKSETZEN' | France: 'Remise a Zero' | English: 'RESET'
  281 = 'Reset Done' | German: 'ZURUCKSETZEN  ABGESCHLOSSEN' | France: 'REMISE TERMINE' | English: 'Reset Done'
  1405 = 'RESET REMAINING\nDOSING TOTALIZER (ml)' | German: 'RÜCKSTELLUNG DER\nRESTDOSIERUNG TOTALIZER (ml)' | France: 'RESET TOTALISATEUR DE\nDOSES RESTANTES (ml)' | English: 'RESET REMAINING\nDOSING TOTALIZER (ml)'
